(* IEC 61131-3 sources: CodesysTest/export (part 2) *)

(* ---- FB_CollectionHandlerAll.st ---- *)
FUNCTION_BLOCK FINAL FB_CollectionHandlerAll
VAR_INPUT
END_VAR
VAR
	Collection: ARRAY[0..GlobalObjects.MAX_OBJECTS] OF IAllObjects; // object array
	ObjNames   : ARRAY[0..GlobalObjects.MAX_OBJECTS] OF STRING;
	_ArrayOver   : BOOL;
	_BadObj      : INT;
	_DupeObj   : INT;
	_OverObj   : INT;
	_TotalObj   : UINT;
END_VAR

METHOD FINAL AddObject
VAR_INPUT
	Obj   : IAllObjects;
END_VAR
VAR
	AnyObject : IAllObjects;
	Fault : IFault;
	Cylinder : ICylinder;
	PositionableMotor : IPositionableMotor;
	Logger : IMachineLogger;
	Loggable : ILoggable;
	Executable : IExecuteAutomatically;
	Initializable : IInitializable;
	J   : UINT;
END_VAR
IF (__QUERYINTERFACE(Obj, AnyObject)) THEN
   // make sure haven't already added this object
   FOR J:= 1 TO _TotalObj DO
      IF Collection[J] = AnyObject THEN
         // object pointer matches - dupe!
         _DupeObj:= _DupeObj + 1;
         RETURN;
      END_IF
   END_FOR

   IF _TotalObj < GlobalObjects.MAX_OBJECTS THEN
      Collection[_TotalObj]:= AnyObject;
      ObjNames[_TotalObj]:= Obj.InstanceName;
	   _TotalObj:= _TotalObj + 1;
   ELSE
      _ArrayOver:= TRUE;
      _OverObj:= _OverObj + 1;
   END_IF
ELSE
   _BadObj:= _BadObj + 1;
END_IF

// Add object to proper collection based on its interfaces
IF (__QUERYINTERFACE(Obj, Fault)) THEN
	GlobalObjects.CollectionOfFaults.AddObject(Fault);
END_IF

IF (__QUERYINTERFACE(Obj, Cylinder)) THEN
	GlobalObjects.CollectionOfCylinders.AddObject(Cylinder);
END_IF

IF (__QUERYINTERFACE(Obj, PositionableMotor)) THEN
	GlobalObjects.CollectionOfPositionableMotors.AddObject(PositionableMotor);
END_IF

IF (__QUERYINTERFACE(Obj, Logger)) THEN
	GlobalObjects.CollectionOfLogs.AddObject(Logger);
END_IF

IF (__QUERYINTERFACE(Obj, Loggable)) THEN
	GlobalObjects.CollectionOfLoggable.AddObject(Loggable);
END_IF

IF (__QUERYINTERFACE(Obj, Executable)) THEN
	GlobalObjects.CollectionOfExecutable.AddObject(Executable);
END_IF

IF (__QUERYINTERFACE(Obj, Initializable)) THEN
	GlobalObjects.CollectionOfInitialzable.AddObject(Initializable);
END_IF

FUNCTION_BLOCK FINAL FB_CollectionHandlerAll
VAR_INPUT
END_VAR
VAR
	Collection: ARRAY[0..GlobalObjects.MAX_OBJECTS] OF IAllObjects; // object array
	ObjNames   : ARRAY[0..GlobalObjects.MAX_OBJECTS] OF STRING;
	_ArrayOver   : BOOL;
	_BadObj      : INT;
	_DupeObj   : INT;
	_OverObj   : INT;
	_TotalObj   : UINT;
END_VAR

METHOD FINAL AddObject
VAR_INPUT
	Obj   : IAllObjects;
END_VAR
VAR
	AnyObject : IAllObjects;
	Fault : IFault;
	Cylinder : ICylinder;
	PositionableMotor : IPositionableMotor;
	Logger : IMachineLogger;
	Loggable : ILoggable;
	Executable : IExecuteAutomatically;
	Initializable : IInitializable;
	J   : UINT;
END_VAR
IF (__QUERYINTERFACE(Obj, AnyObject)) THEN
   // make sure haven't already added this object
   FOR J:= 1 TO _TotalObj DO
      IF Collection[J] = AnyObject THEN
         // object pointer matches - dupe!
         _DupeObj:= _DupeObj + 1;
         RETURN;
      END_IF
   END_FOR

   IF _TotalObj < GlobalObjects.MAX_OBJECTS THEN
      Collection[_TotalObj]:= AnyObject;
      ObjNames[_TotalObj]:= Obj.InstanceName;
	   _TotalObj:= _TotalObj + 1;
   ELSE
      _ArrayOver:= TRUE;
      _OverObj:= _OverObj + 1;
   END_IF
ELSE
   _BadObj:= _BadObj + 1;
END_IF

// Add object to proper collection based on its interfaces
IF (__QUERYINTERFACE(Obj, Fault)) THEN
	GlobalObjects.CollectionOfFaults.AddObject(Fault);
END_IF

IF (__QUERYINTERFACE(Obj, Cylinder)) THEN
	GlobalObjects.CollectionOfCylinders.AddObject(Cylinder);
END_IF

IF (__QUERYINTERFACE(Obj, PositionableMotor)) THEN
	GlobalObjects.CollectionOfPositionableMotors.AddObject(PositionableMotor);
END_IF

IF (__QUERYINTERFACE(Obj, Logger)) THEN
	GlobalObjects.CollectionOfLogs.AddObject(Logger);
END_IF

IF (__QUERYINTERFACE(Obj, Loggable)) THEN
	GlobalObjects.CollectionOfLoggable.AddObject(Loggable);
END_IF

IF (__QUERYINTERFACE(Obj, Executable)) THEN
	GlobalObjects.CollectionOfExecutable.AddObject(Executable);
END_IF

IF (__QUERYINTERFACE(Obj, Initializable)) THEN
	GlobalObjects.CollectionOfInitialzable.AddObject(Initializable);
END_IF

(* ---- FB_CollectionHandlerCylinders.st ---- *)
FUNCTION_BLOCK FB_CollectionHandlerCylinders
VAR_INPUT
END_VAR
VAR
	Collection: ARRAY[0..GlobalObjects.MAX_CYLINDERS] OF ICylinder; // object array
	ObjNames   : ARRAY[0..GlobalObjects.MAX_CYLINDERS] OF STRING;
	_ArrayOver   : BOOL;
	_BadObj      : INT;
	_DupeObj   : INT;
	_OverObj   : INT;
	_TotalObj   : UINT;
END_VAR

METHOD AddObject
VAR_INPUT
	Obj   : ICylinder;
END_VAR
VAR
	Cast: ICylinder;
	J   : UINT;
END_VAR
FOR J:= 0 TO _TotalObj DO
	IF Collection[J] = Obj THEN
		// object pointer matches - dupe!
		_DupeObj:= _DupeObj + 1;
		RETURN;
	END_IF
END_FOR

IF _TotalObj < GlobalObjects.MAX_CYLINDERS THEN
	Collection[_TotalObj]:= Obj;
	ObjNames[_TotalObj]:= Obj.InstanceName;
	_TotalObj:= _TotalObj + 1;
ELSE
	_ArrayOver:= TRUE;
	_OverObj:= _OverObj + 1;
END_IF

FUNCTION_BLOCK FB_CollectionHandlerCylinders
VAR_INPUT
END_VAR
VAR
	Collection: ARRAY[0..GlobalObjects.MAX_CYLINDERS] OF ICylinder; // object array
	ObjNames   : ARRAY[0..GlobalObjects.MAX_CYLINDERS] OF STRING;
	_ArrayOver   : BOOL;
	_BadObj      : INT;
	_DupeObj   : INT;
	_OverObj   : INT;
	_TotalObj   : UINT;
END_VAR

METHOD AddObject
VAR_INPUT
	Obj   : ICylinder;
END_VAR
VAR
	Cast: ICylinder;
	J   : UINT;
END_VAR
FOR J:= 0 TO _TotalObj DO
	IF Collection[J] = Obj THEN
		// object pointer matches - dupe!
		_DupeObj:= _DupeObj + 1;
		RETURN;
	END_IF
END_FOR

IF _TotalObj < GlobalObjects.MAX_CYLINDERS THEN
	Collection[_TotalObj]:= Obj;
	ObjNames[_TotalObj]:= Obj.InstanceName;
	_TotalObj:= _TotalObj + 1;
ELSE
	_ArrayOver:= TRUE;
	_OverObj:= _OverObj + 1;
END_IF

(* ---- FB_CollectionHandlerExecutable.st ---- *)
FUNCTION_BLOCK FB_CollectionHandlerExecutable
VAR_INPUT
END_VAR
VAR
	Collection: ARRAY[0..GlobalObjects.MAX_EXECUTEABLE] OF IExecuteAutomatically; // object array
	ObjNames   : ARRAY[0..GlobalObjects.MAX_EXECUTEABLE] OF STRING;
	_ArrayOver   : BOOL;
	_BadObj      : INT;
	_DupeObj   : INT;
	_OverObj   : INT;
	_TotalObj   : UINT;
END_VAR
//	Function Block: FB_CollectionHandlerExecutable
//	Description: This collection handler stores executable FB's to an array
//				 and has a method to execute them all on demand
//	Created by: Ben Hess
//	Created Date: Friday, September 7, 2018

METHOD AddObject
VAR_INPUT
	Obj   : IExecuteAutomatically;
END_VAR
VAR
	I   : UINT;
	J : UINT;
END_VAR
// Add the active fault to the array
FOR J:= 0 TO _TotalObj DO
	IF Collection[J] = Obj THEN
		// object pointer matches - it's already in here
		RETURN;
	END_IF
END_FOR

IF _TotalObj < GlobalObjects.MAX_EXECUTEABLE THEN
	Collection[_TotalObj]:= Obj;
	ObjNames[_TotalObj]:= Obj.InstanceName;
	_TotalObj:= _TotalObj + 1;
ELSE
	_ArrayOver:= TRUE;
	_OverObj:= _OverObj + 1;
END_IF

METHOD ExecuteAll
VAR_INPUT
END_VAR
VAR
	Cast : IExecuteAutomatically;
	J : UINT;
END_VAR
// For each executable objest in the array, run its "Execute()" method
FOR J:= 0 TO _TotalObj - 1 DO
	IF (__QUERYINTERFACE(Collection[J], Cast)) THEN
		Cast.Execute();
	ELSE
		RETURN;
	END_IF
END_FOR

FUNCTION_BLOCK FB_CollectionHandlerExecutable
VAR_INPUT
END_VAR
VAR
	Collection: ARRAY[0..GlobalObjects.MAX_EXECUTEABLE] OF IExecuteAutomatically; // object array
	ObjNames   : ARRAY[0..GlobalObjects.MAX_EXECUTEABLE] OF STRING;
	_ArrayOver   : BOOL;
	_BadObj      : INT;
	_DupeObj   : INT;
	_OverObj   : INT;
	_TotalObj   : UINT;
END_VAR
//	Function Block: FB_CollectionHandlerExecutable
//	Description: This collection handler stores executable FB's to an array
//				 and has a method to execute them all on demand
//	Created by: Ben Hess
//	Created Date: Friday, September 7, 2018

METHOD AddObject
VAR_INPUT
	Obj   : IExecuteAutomatically;
END_VAR
VAR
	I   : UINT;
	J : UINT;
END_VAR
// Add the active fault to the array
FOR J:= 0 TO _TotalObj DO
	IF Collection[J] = Obj THEN
		// object pointer matches - it's already in here
		RETURN;
	END_IF
END_FOR

IF _TotalObj < GlobalObjects.MAX_EXECUTEABLE THEN
	Collection[_TotalObj]:= Obj;
	ObjNames[_TotalObj]:= Obj.InstanceName;
	_TotalObj:= _TotalObj + 1;
ELSE
	_ArrayOver:= TRUE;
	_OverObj:= _OverObj + 1;
END_IF

METHOD ExecuteAll
VAR_INPUT
END_VAR
VAR
	Cast : IExecuteAutomatically;
	J : UINT;
END_VAR
// For each executable objest in the array, run its "Execute()" method
FOR J:= 0 TO _TotalObj - 1 DO
	IF (__QUERYINTERFACE(Collection[J], Cast)) THEN
		Cast.Execute();
	ELSE
		RETURN;
	END_IF
END_FOR

(* ---- FB_CollectionHandlerFaults.st ---- *)
FUNCTION_BLOCK FB_CollectionHandlerFaults
VAR_INPUT
END_VAR
VAR
	Collection: ARRAY[0..GlobalObjects.MAX_FAULTS] OF IFault; // object array
	ObjNames   : ARRAY[0..GlobalObjects.MAX_FAULTS] OF STRING;
	faults : ARRAY[0..GlobalObjects.MAX_FAULTS] OF HMIFaultType;
	_ArrayOver   : BOOL;
	_BadObj      : INT;
	_DupeObj   : INT;
	_OverObj   : INT;
	_TotalObj   : UINT;
	_InitFaultList : BOOL;
END_VAR

METHOD FaultUpdateForHMI
VAR_INPUT
END_VAR
VAR
	I : UINT;
END_VAR
FOR I:= 0 TO _TotalObj - 1 DO
	IF NOT _InitFaultList THEN
		faults[I].name := Collection[I].InstanceName;
	END_IF
	faults[I].active := Collection[I].FaultActive;
END_FOR
_InitFaultList := TRUE;

METHOD AddObject
VAR_INPUT
	Obj   : IFault;
END_VAR
VAR
	J   : UINT;
END_VAR
FOR J:= 0 TO _TotalObj DO
	IF Collection[J] = Obj THEN
		// object pointer matches - dupe!
		_DupeObj:= _DupeObj + 1;
		RETURN;
	END_IF
END_FOR

IF _TotalObj < GlobalObjects.MAX_FAULTS THEN
	Collection[_TotalObj]:= Obj;
	ObjNames[_TotalObj]:= Obj.InstanceName;
	_TotalObj:= _TotalObj + 1;
ELSE
	_ArrayOver:= TRUE;
	_OverObj:= _OverObj + 1;
END_IF

(* ---- FB_CollectionHandlerInitializable.st ---- *)
FUNCTION_BLOCK FB_CollectionHandlerInitializable
VAR_INPUT

END_VAR
VAR
	Collection: ARRAY[0..GlobalObjects.MAX_LOGGABLE] OF IInitializable; // object array
	ObjNames   : ARRAY[0..GlobalObjects.MAX_LOGGABLE] OF STRING;
	_ArrayOver   : BOOL;
	_BadObj      : INT;
	_DupeObj   : INT;
	_OverObj   : INT;
	_TotalObj   : UINT;
END_VAR
//	Function Block: FB_CollectionHandlerLoggable
//	Description: This collection handler takes in loggable objects and registers them with a logger.  The FirstScan function should trigger the
//				 RegisterAll() method to register all loggable objects with a logger
//	Created by: Ben Hess
//	Created Date: Tuesday, September 11, 2018

METHOD AddObject
VAR_INPUT
	Obj   : IInitializable;
END_VAR
VAR
	J   : UINT;
END_VAR
FOR J:= 0 TO _TotalObj DO
	IF Collection[J] = Obj THEN
		// object pointer matches - dupe!
		_DupeObj:= _DupeObj + 1;
		RETURN;
	END_IF
END_FOR

IF _TotalObj < GlobalObjects.MAX_LOGGABLE THEN
	Collection[_TotalObj]:= Obj;
	ObjNames[_TotalObj]:= Obj.InstanceName;
	_TotalObj:= _TotalObj + 1;
ELSE
	_ArrayOver:= TRUE;
	_OverObj:= _OverObj + 1;
END_IF

METHOD InitializeAll
VAR_INPUT

END_VAR
VAR
	J : UINT;
	Cast : IInitializable;
END_VAR

FOR J:= 0 TO _TotalObj - 1 DO
	IF (__QUERYINTERFACE(Collection[J], Cast)) THEN
		Cast.Initialize();
	ELSE
		RETURN;
	END_IF
END_FOR

FUNCTION_BLOCK FB_CollectionHandlerInitializable
VAR_INPUT

END_VAR
VAR
	Collection: ARRAY[0..GlobalObjects.MAX_LOGGABLE] OF IInitializable; // object array
	ObjNames   : ARRAY[0..GlobalObjects.MAX_LOGGABLE] OF STRING;
	_ArrayOver   : BOOL;
	_BadObj      : INT;
	_DupeObj   : INT;
	_OverObj   : INT;
	_TotalObj   : UINT;
END_VAR
//	Function Block: FB_CollectionHandlerLoggable
//	Description: This collection handler takes in loggable objects and registers them with a logger.  The FirstScan function should trigger the
//				 RegisterAll() method to register all loggable objects with a logger
//	Created by: Ben Hess
//	Created Date: Tuesday, September 11, 2018

METHOD AddObject
VAR_INPUT
	Obj   : IInitializable;
END_VAR
VAR
	J   : UINT;
END_VAR
FOR J:= 0 TO _TotalObj DO
	IF Collection[J] = Obj THEN
		// object pointer matches - dupe!
		_DupeObj:= _DupeObj + 1;
		RETURN;
	END_IF
END_FOR

IF _TotalObj < GlobalObjects.MAX_LOGGABLE THEN
	Collection[_TotalObj]:= Obj;
	ObjNames[_TotalObj]:= Obj.InstanceName;
	_TotalObj:= _TotalObj + 1;
ELSE
	_ArrayOver:= TRUE;
	_OverObj:= _OverObj + 1;
END_IF

METHOD InitializeAll
VAR_INPUT

END_VAR
VAR
	J : UINT;
	Cast : IInitializable;
END_VAR

FOR J:= 0 TO _TotalObj - 1 DO
	IF (__QUERYINTERFACE(Collection[J], Cast)) THEN
		Cast.Initialize();
	ELSE
		RETURN;
	END_IF
END_FOR

(* ---- FB_CollectionHandlerLoggable.st ---- *)
FUNCTION_BLOCK FB_CollectionHandlerLoggable
VAR_INPUT

END_VAR
VAR
	Collection: ARRAY[0..GlobalObjects.MAX_LOGGABLE] OF ILoggable; // object array
	ObjNames   : ARRAY[0..GlobalObjects.MAX_LOGGABLE] OF STRING;
	_ArrayOver   : BOOL;
	_BadObj      : INT;
	_DupeObj   : INT;
	_OverObj   : INT;
	_TotalObj   : UINT;
	_internalLogger : REFERENCE TO IMachineLogger;
END_VAR
//	Function Block: FB_CollectionHandlerLoggable
//	Description: This collection handler takes in loggable objects and registers them with a logger.  The FirstScan function should trigger the
//				 RegisterAll() method to register all loggable objects with a logger
//	Created by: Ben Hess
//	Created Date: Tuesday, September 11, 2018

METHOD AddObject
VAR_INPUT
	Obj   : ILoggable;
END_VAR
VAR
	J   : UINT;
END_VAR
FOR J:= 0 TO _TotalObj DO
	IF Collection[J] = Obj THEN
		// object pointer matches - dupe!
		_DupeObj:= _DupeObj + 1;
		RETURN;
	END_IF
END_FOR

IF _TotalObj < GlobalObjects.MAX_LOGGABLE THEN
	Collection[_TotalObj]:= Obj;
	ObjNames[_TotalObj]:= Obj.InstanceName;
	_TotalObj:= _TotalObj + 1;
ELSE
	_ArrayOver:= TRUE;
	_OverObj:= _OverObj + 1;
END_IF

METHOD RegisterAll
VAR_INPUT
	internalLogger : IMachineLogger;
END_VAR
VAR
	I   : UINT;
	J : UINT;
	cast : ILoggable;
END_VAR

FOR J:= 0 TO _TotalObj - 1 DO
	IF (__QUERYINTERFACE(Collection[J], Cast)) THEN
		cast.RegisterLogger(internalLogger := internalLogger);
	ELSE
		RETURN;
	END_IF
END_FOR

FUNCTION_BLOCK FB_CollectionHandlerLoggable
VAR_INPUT

END_VAR
VAR
	Collection: ARRAY[0..GlobalObjects.MAX_LOGGABLE] OF ILoggable; // object array
	ObjNames   : ARRAY[0..GlobalObjects.MAX_LOGGABLE] OF STRING;
	_ArrayOver   : BOOL;
	_BadObj      : INT;
	_DupeObj   : INT;
	_OverObj   : INT;
	_TotalObj   : UINT;
	_internalLogger : REFERENCE TO IMachineLogger;
END_VAR
//	Function Block: FB_CollectionHandlerLoggable
//	Description: This collection handler takes in loggable objects and registers them with a logger.  The FirstScan function should trigger the
//				 RegisterAll() method to register all loggable objects with a logger
//	Created by: Ben Hess
//	Created Date: Tuesday, September 11, 2018

METHOD AddObject
VAR_INPUT
	Obj   : ILoggable;
END_VAR
VAR
	J   : UINT;
END_VAR
FOR J:= 0 TO _TotalObj DO
	IF Collection[J] = Obj THEN
		// object pointer matches - dupe!
		_DupeObj:= _DupeObj + 1;
		RETURN;
	END_IF
END_FOR

IF _TotalObj < GlobalObjects.MAX_LOGGABLE THEN
	Collection[_TotalObj]:= Obj;
	ObjNames[_TotalObj]:= Obj.InstanceName;
	_TotalObj:= _TotalObj + 1;
ELSE
	_ArrayOver:= TRUE;
	_OverObj:= _OverObj + 1;
END_IF

METHOD RegisterAll
VAR_INPUT
	internalLogger : IMachineLogger;
END_VAR
VAR
	I   : UINT;
	J : UINT;
	cast : ILoggable;
END_VAR

FOR J:= 0 TO _TotalObj - 1 DO
	IF (__QUERYINTERFACE(Collection[J], Cast)) THEN
		cast.RegisterLogger(internalLogger := internalLogger);
	ELSE
		RETURN;
	END_IF
END_FOR

(* ---- FB_CollectionHandlerLogs.st ---- *)
FUNCTION_BLOCK FB_CollectionHandlerLogs
VAR_INPUT
END_VAR
VAR
	Collection: ARRAY[0..GlobalObjects.MAX_LOGS] OF IMachineLogger; // object array
	ObjNames   : ARRAY[0..GlobalObjects.MAX_LOGS] OF STRING;
	_ArrayOver   : BOOL;
	_BadObj      : INT;
	_DupeObj   : INT;
	_OverObj   : INT;
	_TotalObj   : UINT;
END_VAR

METHOD AddObject
VAR_INPUT
	Obj   : IMachineLogger;
END_VAR
VAR
	J   : UINT;
END_VAR
FOR J:= 0 TO _TotalObj DO
	IF Collection[J] = Obj THEN
		// object pointer matches - dupe!
		_DupeObj:= _DupeObj + 1;
		RETURN;
	END_IF
END_FOR

IF _TotalObj < GlobalObjects.MAX_LOGS THEN
	Collection[_TotalObj]:= Obj;
	ObjNames[_TotalObj]:= Obj.InstanceName;
	_TotalObj:= _TotalObj + 1;
ELSE
	_ArrayOver:= TRUE;
	_OverObj:= _OverObj + 1;
END_IF

(* ---- FB_CollectionHandlerPositionableMotors.st ---- *)
FUNCTION_BLOCK FB_CollectionHandlerPositionableMotors
VAR_INPUT
END_VAR
VAR
	Collection: ARRAY[0..GlobalObjects.MAX_MOTORS] OF IPositionableMotor; // object array
	ObjNames   : ARRAY[0..GlobalObjects.MAX_MOTORS] OF STRING;
	_ArrayOver   : BOOL;
	_BadObj      : INT;
	_DupeObj   : INT;
	_OverObj   : INT;
	_TotalObj   : UINT;
END_VAR

METHOD AddObject
VAR_INPUT
	Obj   : IPositionableMotor;
END_VAR
VAR
	J   : UINT;
END_VAR
FOR J:= 0 TO _TotalObj DO
	IF Collection[J] = Obj THEN
		// object pointer matches - dupe!
		_DupeObj:= _DupeObj + 1;
		RETURN;
	END_IF
END_FOR

IF _TotalObj < GlobalObjects.MAX_MOTORS THEN
	Collection[_TotalObj]:= Obj;
	ObjNames[_TotalObj]:= Obj.InstanceName;
	_TotalObj:= _TotalObj + 1;
ELSE
	_ArrayOver:= TRUE;
	_OverObj:= _OverObj + 1;
END_IF

FUNCTION_BLOCK FB_CollectionHandlerPositionableMotors
VAR_INPUT
END_VAR
VAR
	Collection: ARRAY[0..GlobalObjects.MAX_MOTORS] OF IPositionableMotor; // object array
	ObjNames   : ARRAY[0..GlobalObjects.MAX_MOTORS] OF STRING;
	_ArrayOver   : BOOL;
	_BadObj      : INT;
	_DupeObj   : INT;
	_OverObj   : INT;
	_TotalObj   : UINT;
END_VAR

METHOD AddObject
VAR_INPUT
	Obj   : IPositionableMotor;
END_VAR
VAR
	J   : UINT;
END_VAR
FOR J:= 0 TO _TotalObj DO
	IF Collection[J] = Obj THEN
		// object pointer matches - dupe!
		_DupeObj:= _DupeObj + 1;
		RETURN;
	END_IF
END_FOR

IF _TotalObj < GlobalObjects.MAX_MOTORS THEN
	Collection[_TotalObj]:= Obj;
	ObjNames[_TotalObj]:= Obj.InstanceName;
	_TotalObj:= _TotalObj + 1;
ELSE
	_ArrayOver:= TRUE;
	_OverObj:= _OverObj + 1;
END_IF

(* ---- FB_Delay.st ---- *)
FUNCTION_BLOCK FB_Delay IMPLEMENTS IExecuteAutomatically
VAR_INPUT
	in : BOOL;
	delay : TIME;
END_VAR
VAR_OUTPUT
	Q : BOOL;
END_VAR
VAR
	delayTimer : TON;
END_VAR

METHOD Execute

delayTimer(IN := in, PT := delay, Q => Q);

FUNCTION_BLOCK FB_Delay IMPLEMENTS IExecuteAutomatically
VAR_INPUT
	in : BOOL;
	delay : TIME;
END_VAR
VAR_OUTPUT
	Q : BOOL;
END_VAR
VAR
	delayTimer : TON;
END_VAR

METHOD Execute

delayTimer(IN := in, PT := delay, Q => Q);

(* ---- FB_DoubleSolenoidClosedCenterActuator.st ---- *)
FUNCTION_BLOCK FB_DoubleSolenoidClosedCenterActuator EXTENDS FB_PneumaticActuator IMPLEMENTS IExtendLowPressure
VAR_INPUT
END_VAR
VAR_OUTPUT
END_VAR
VAR

END_VAR

PROPERTY ExtendAsserted : BOOL

PROPERTY RetractAsserted : BOOL

METHOD Extend

THIS^.solenoid0 := TRUE;
THIS^.solenoid1 := FALSE;

METHOD Retract

THIS^.solenoid0 := FALSE;
THIS^.solenoid1 := TRUE;

METHOD ExtendLowPressure
VAR_INPUT
END_VAR

THIS^.solenoid0 := TRUE;
THIS^.solenoid1 := TRUE;

PROPERTY ExtendLPAsserted : BOOL

FUNCTION_BLOCK FB_DoubleSolenoidClosedCenterActuator EXTENDS FB_PneumaticActuator IMPLEMENTS IExtendLowPressure
VAR_INPUT
END_VAR
VAR_OUTPUT
END_VAR
VAR

END_VAR

PROPERTY ExtendAsserted : BOOL

PROPERTY RetractAsserted : BOOL

METHOD Extend

THIS^.solenoid0 := TRUE;
THIS^.solenoid1 := FALSE;

METHOD Retract

THIS^.solenoid0 := FALSE;
THIS^.solenoid1 := TRUE;

METHOD ExtendLowPressure
VAR_INPUT
END_VAR

THIS^.solenoid0 := TRUE;
THIS^.solenoid1 := TRUE;

PROPERTY ExtendLPAsserted : BOOL

(* ---- FB_DoubleSolenoidClosedCenterActuator_UnitTests.st ---- *)
(*
*)
{attribute 'test' := 'multitest'}
{attribute 'testcasename':='Double Solenoid Closed Center'}
{attribute 'testcategory':='Solenoids'}
{attribute 'testcasetimeout':='15000'}
FUNCTION_BLOCK FB_DoubleSolenoidClosedCenterActuator_UnitTests EXTENDS CBM.EtrigA
VAR_INPUT
	xGetTestInfo : BOOL;
    diTestCaseIndex : DINT;
END_VAR
VAR_OUTPUT
    sTestCaseName : STRING;
	sTestCaseCategories : STRING;
    diTestCaseCount : DINT;
    diTestCaseTimeout : DINT;
    sInfo : STRING;
	eError : UnitTestErrors;
    sError : STRING;
    eFailureMode : TM.FAILUREMODE;
END_VAR
VAR
	testee : FB_DoubleSolenoidClosedCenterActuator(name := 'Unit Test Actuator');
END_VAR
SUPER^();

{attribute 'hide'}
METHOD prvAbort : BOOL

SUPER^.prvAbort();

xAbortInProgress := FALSE;

{attribute 'hide'}
METHOD prvCyclicAction : BOOL

SUPER^.prvCyclicAction();
THIS^.diTestCaseCount := 4;

CASE diTestCaseIndex OF
    0: // Test Case #0
        IF THIS^.xGetTestInfo THEN
            THIS^.sTestCaseName := 'Step 1: Test Solonoids Off';
            THIS^.sTestCaseCategories := 'Solenoids';
            THIS^.diTestCaseTimeout := 3000;
			xDone := TRUE;
		ELSE
			IF NOT testee.Solenoid0Asserted AND NOT testee.Solenoid1Asserted THEN
				 xDone := TRUE;
			ELSE
				THIS^.sError := 'Solenoids not off';
				xError := TRUE;
				eError := UnitTestErrors.Failure;
            	eFailureMode := TM.FAILUREMODE.AbortTestCase;
                iError := 1;
			END_IF
        END_IF
    1: // Test Case #1
        IF THIS^.xGetTestInfo THEN
            THIS^.sTestCaseName := 'Step 2: Extend Cylinder';
            THIS^.sTestCaseCategories := 'Solenoids';
            THIS^.diTestCaseTimeout := 3000;
            xDone := TRUE;
		ELSE
			testee.Extend();
			IF testee.Solenoid0Asserted AND testee.ExtendAsserted
				AND NOT testee.Solenoid1Asserted AND NOT testee.RetractAsserted THEN
				 xDone := TRUE;
			ELSE
				THIS^.sError := 'Failed to extend';
				xError := TRUE;
				eError := UnitTestErrors.Failure;
            	eFailureMode := TM.FAILUREMODE.AbortTestCase;
                iError := 2;
			END_IF
       END_IF

	2:	//
		IF THIS^.xGetTestInfo THEN
            THIS^.sTestCaseName := 'Step 3: Retract Cylinder';
            THIS^.sTestCaseCategories := 'Solenoids';
            THIS^.diTestCaseTimeout := 3000;
            xDone := TRUE;
		ELSE
			testee.Retract();
			IF testee.Solenoid1Asserted AND testee.RetractAsserted
				AND NOT testee.Solenoid0Asserted AND NOT testee.ExtendAsserted THEN
				 xDone := TRUE;
			ELSE
				THIS^.sError := 'Failed to retract';
				xError := TRUE;
				eError := UnitTestErrors.Failure;
            	eFailureMode := TM.FAILUREMODE.AbortTestCase;
                iError := 3;
			END_IF
       END_IF

   	3:	IF THIS^.xGetTestInfo THEN
            THIS^.sTestCaseName := 'Step 4: Extend Low Pressure';
            THIS^.sTestCaseCategories := 'Solenoids';
            THIS^.diTestCaseTimeout := 3000;
            xDone := TRUE;
		ELSE
			testee.ExtendLowPressure();
			IF testee.Solenoid1Asserted AND testee.ExtendLPAsserted
				AND testee.Solenoid0Asserted
				AND NOT testee.RetractAsserted THEN
				 xDone := TRUE;
			ELSE
				THIS^.sError := 'Failed to extend low pressure';
				xError := TRUE;
				eError := UnitTestErrors.Failure;
            	eFailureMode := TM.FAILUREMODE.AbortTestCase;
                iError := 3;
			END_IF
       END_IF
    ELSE
        IF THIS^.diTestCaseIndex < 0 THEN
            THIS^.diTestCaseCount := 4;
            xDone := TRUE;
        ELSE
            THIS^.sInfo := 'Invalid test case index';
            eError := UnitTestErrors.Failure;
			xError := TRUE;
        END_IF
END_CASE

{attribute 'hide'}
METHOD prvResetOutputs : BOOL

SUPER^.prvResetOutputs();

sTestCaseName := '';
sTestCaseCategories := '';
diTestCaseCount := 0;
diTestCaseTimeout := 0;
sInfo := '';
sError := '';
eFailureMode := TM.FAILUREMODE.AbortTestCase;

{attribute 'hide'}
METHOD prvStart : BOOL

SUPER^.prvStart();

(*
*)
{attribute 'test' := 'multitest'}
{attribute 'testcasename':='Double Solenoid Closed Center'}
{attribute 'testcategory':='Solenoids'}
{attribute 'testcasetimeout':='15000'}
FUNCTION_BLOCK FB_DoubleSolenoidClosedCenterActuator_UnitTests EXTENDS CBM.EtrigA
VAR_INPUT
	xGetTestInfo : BOOL;
    diTestCaseIndex : DINT;
END_VAR
VAR_OUTPUT
    sTestCaseName : STRING;
	sTestCaseCategories : STRING;
    diTestCaseCount : DINT;
    diTestCaseTimeout : DINT;
    sInfo : STRING;
	eError : UnitTestErrors;
    sError : STRING;
    eFailureMode : TM.FAILUREMODE;
END_VAR
VAR
	testee : FB_DoubleSolenoidClosedCenterActuator(name := 'Unit Test Actuator');
END_VAR
SUPER^();

{attribute 'hide'}
METHOD prvAbort : BOOL

SUPER^.prvAbort();

xAbortInProgress := FALSE;

{attribute 'hide'}
METHOD prvCyclicAction : BOOL

SUPER^.prvCyclicAction();
THIS^.diTestCaseCount := 4;

CASE diTestCaseIndex OF
    0: // Test Case #0
        IF THIS^.xGetTestInfo THEN
            THIS^.sTestCaseName := 'Step 1: Test Solonoids Off';
            THIS^.sTestCaseCategories := 'Solenoids';
            THIS^.diTestCaseTimeout := 3000;
			xDone := TRUE;
		ELSE
			IF NOT testee.Solenoid0Asserted AND NOT testee.Solenoid1Asserted THEN
				 xDone := TRUE;
			ELSE
				THIS^.sError := 'Solenoids not off';
				xError := TRUE;
				eError := UnitTestErrors.Failure;
            	eFailureMode := TM.FAILUREMODE.AbortTestCase;
                iError := 1;
			END_IF
        END_IF
    1: // Test Case #1
        IF THIS^.xGetTestInfo THEN
            THIS^.sTestCaseName := 'Step 2: Extend Cylinder';
            THIS^.sTestCaseCategories := 'Solenoids';
            THIS^.diTestCaseTimeout := 3000;
            xDone := TRUE;
		ELSE
			testee.Extend();
			IF testee.Solenoid0Asserted AND testee.ExtendAsserted
				AND NOT testee.Solenoid1Asserted AND NOT testee.RetractAsserted THEN
				 xDone := TRUE;
			ELSE
				THIS^.sError := 'Failed to extend';
				xError := TRUE;
				eError := UnitTestErrors.Failure;
            	eFailureMode := TM.FAILUREMODE.AbortTestCase;
                iError := 2;
			END_IF
       END_IF

	2:	//
		IF THIS^.xGetTestInfo THEN
            THIS^.sTestCaseName := 'Step 3: Retract Cylinder';
            THIS^.sTestCaseCategories := 'Solenoids';
            THIS^.diTestCaseTimeout := 3000;
            xDone := TRUE;
		ELSE
			testee.Retract();
			IF testee.Solenoid1Asserted AND testee.RetractAsserted
				AND NOT testee.Solenoid0Asserted AND NOT testee.ExtendAsserted THEN
				 xDone := TRUE;
			ELSE
				THIS^.sError := 'Failed to retract';
				xError := TRUE;
				eError := UnitTestErrors.Failure;
            	eFailureMode := TM.FAILUREMODE.AbortTestCase;
                iError := 3;
			END_IF
       END_IF

   	3:	IF THIS^.xGetTestInfo THEN
            THIS^.sTestCaseName := 'Step 4: Extend Low Pressure';
            THIS^.sTestCaseCategories := 'Solenoids';
            THIS^.diTestCaseTimeout := 3000;
            xDone := TRUE;
		ELSE
			testee.ExtendLowPressure();
			IF testee.Solenoid1Asserted AND testee.ExtendLPAsserted
				AND testee.Solenoid0Asserted
				AND NOT testee.RetractAsserted THEN
				 xDone := TRUE;
			ELSE
				THIS^.sError := 'Failed to extend low pressure';
				xError := TRUE;
				eError := UnitTestErrors.Failure;
            	eFailureMode := TM.FAILUREMODE.AbortTestCase;
                iError := 3;
			END_IF
       END_IF
    ELSE
        IF THIS^.diTestCaseIndex < 0 THEN
            THIS^.diTestCaseCount := 4;
            xDone := TRUE;
        ELSE
            THIS^.sInfo := 'Invalid test case index';
            eError := UnitTestErrors.Failure;
			xError := TRUE;
        END_IF
END_CASE

{attribute 'hide'}
METHOD prvResetOutputs : BOOL

SUPER^.prvResetOutputs();

sTestCaseName := '';
sTestCaseCategories := '';
diTestCaseCount := 0;
diTestCaseTimeout := 0;
sInfo := '';
sError := '';
eFailureMode := TM.FAILUREMODE.AbortTestCase;

{attribute 'hide'}
METHOD prvStart : BOOL

SUPER^.prvStart();

(* ---- FB_DoubleSolenoidOpenCenterActuator.st ---- *)
FUNCTION_BLOCK FINAL FB_DoubleSolenoidOpenCenterActuator EXTENDS FB_DoubleSolenoidClosedCenterActuator IMPLEMENTS IExhaustable
VAR_INPUT
END_VAR
VAR_OUTPUT
END_VAR
VAR
END_VAR

METHOD Exhaust : BOOL

THIS^.solenoid0 := FALSE;
THIS^.solenoid1 := FALSE;

FUNCTION_BLOCK FINAL FB_DoubleSolenoidOpenCenterActuator EXTENDS FB_DoubleSolenoidClosedCenterActuator IMPLEMENTS IExhaustable
VAR_INPUT
END_VAR
VAR_OUTPUT
END_VAR
VAR
END_VAR

METHOD Exhaust : BOOL

THIS^.solenoid0 := FALSE;
THIS^.solenoid1 := FALSE;

(* ---- FB_DoubleSolenoidOpenCenterActuator_UnitTests.st ---- *)
(*
*)
{attribute 'test' := 'multitest'}
{attribute 'testcasename':='Double Solenoid Open Center'}
{attribute 'testcategory':='Solenoids'}
{attribute 'testcasetimeout':='15000'}
FUNCTION_BLOCK FB_DoubleSolenoidOpenCenterActuator_UnitTests EXTENDS CBM.EtrigA
VAR_INPUT
	xGetTestInfo : BOOL;
    diTestCaseIndex : DINT;
END_VAR
VAR_OUTPUT
    sTestCaseName : STRING;
	sTestCaseCategories : STRING;
    diTestCaseCount : DINT;
    diTestCaseTimeout : DINT;
    sInfo : STRING;
	eError : UnitTestErrors;
    sError : STRING;
    eFailureMode : TM.FAILUREMODE;
END_VAR
VAR
	testee : FB_DoubleSolenoidOpenCenterActuator(name := 'Unit Test Actuator');
END_VAR
SUPER^();

{attribute 'hide'}
METHOD prvAbort : BOOL

SUPER^.prvAbort();

xAbortInProgress := FALSE;

{attribute 'hide'}
METHOD prvCyclicAction : BOOL

SUPER^.prvCyclicAction();
THIS^.diTestCaseCount := 5;

CASE diTestCaseIndex OF
    0: // Test Case #0
        IF THIS^.xGetTestInfo THEN
            THIS^.sTestCaseName := 'Step 1: Test Solonoids Off';
            THIS^.sTestCaseCategories := 'Solenoids';
            THIS^.diTestCaseTimeout := 3000;
			xDone := TRUE;
		ELSE
			IF NOT testee.Solenoid0Asserted AND NOT testee.Solenoid1Asserted THEN
				 xDone := TRUE;
			ELSE
				THIS^.sError := 'Solenoids not off';
				xError := TRUE;
				eError := UnitTestErrors.Failure;
            	eFailureMode := TM.FAILUREMODE.AbortTestCase;
                iError := 1;
			END_IF
        END_IF
    1: // Test Case #1
        IF THIS^.xGetTestInfo THEN
            THIS^.sTestCaseName := 'Step 2: Extend Cylinder';
            THIS^.sTestCaseCategories := 'Solenoids';
            THIS^.diTestCaseTimeout := 3000;
            xDone := TRUE;
		ELSE
			testee.Extend();
			IF testee.Solenoid0Asserted AND testee.ExtendAsserted
				AND NOT testee.Solenoid1Asserted AND NOT testee.RetractAsserted THEN
				 xDone := TRUE;
			ELSE
				THIS^.sError := 'Failed to extend';
				xError := TRUE;
				eError := UnitTestErrors.Failure;
            	eFailureMode := TM.FAILUREMODE.AbortTestCase;
                iError := 2;
			END_IF
       END_IF

	2:	//
		IF THIS^.xGetTestInfo THEN
            THIS^.sTestCaseName := 'Step 3: Retract Cylinder';
            THIS^.sTestCaseCategories := 'Solenoids';
            THIS^.diTestCaseTimeout := 3000;
            xDone := TRUE;
		ELSE
			testee.Retract();
			IF testee.Solenoid1Asserted AND testee.RetractAsserted
				AND NOT testee.Solenoid0Asserted AND NOT testee.ExtendAsserted THEN
				 xDone := TRUE;
			ELSE
				THIS^.sError := 'Failed to retract';
				xError := TRUE;
				eError := UnitTestErrors.Failure;
            	eFailureMode := TM.FAILUREMODE.AbortTestCase;
                iError := 3;
			END_IF
       END_IF

   	3:	IF THIS^.xGetTestInfo THEN
            THIS^.sTestCaseName := 'Step 4: Extend Low Pressure';
            THIS^.sTestCaseCategories := 'Solenoids';
            THIS^.diTestCaseTimeout := 3000;
            xDone := TRUE;
		ELSE
			testee.ExtendLowPressure();
			IF testee.Solenoid1Asserted AND testee.ExtendLPAsserted
				AND testee.Solenoid0Asserted
				AND NOT testee.RetractAsserted THEN
				 xDone := TRUE;
			ELSE
				THIS^.sError := 'Failed to extend low pressure';
				xError := TRUE;
				eError := UnitTestErrors.Failure;
            	eFailureMode := TM.FAILUREMODE.AbortTestCase;
                iError := 3;
			END_IF
       END_IF

	4: // Test Case #4
        IF THIS^.xGetTestInfo THEN
            THIS^.sTestCaseName := 'Step 5: Test Exhaust';
            THIS^.sTestCaseCategories := 'Solenoids';
            THIS^.diTestCaseTimeout := 3000;
			xDone := TRUE;
		ELSE
			testee.Exhaust();
			IF NOT testee.Solenoid0Asserted AND NOT testee.Solenoid1Asserted
				AND NOT testee.ExtendAsserted AND NOT testee.RetractAsserted THEN
				 xDone := TRUE;
			ELSE
				THIS^.sError := 'Solenoids not off';
				xError := TRUE;
				eError := UnitTestErrors.Failure;
            	eFailureMode := TM.FAILUREMODE.AbortTestCase;
                iError := 1;
			END_IF
        END_IF
    ELSE
        IF THIS^.diTestCaseIndex < 0 THEN
            THIS^.diTestCaseCount := 5;
            xDone := TRUE;
        ELSE
            THIS^.sInfo := 'Invalid test case index';
            eError := UnitTestErrors.Failure;
			xError := TRUE;
        END_IF
END_CASE

{attribute 'hide'}
METHOD prvResetOutputs : BOOL

SUPER^.prvResetOutputs();

sTestCaseName := '';
sTestCaseCategories := '';
diTestCaseCount := 0;
diTestCaseTimeout := 0;
sInfo := '';
sError := '';
eFailureMode := TM.FAILUREMODE.AbortTestCase;

{attribute 'hide'}
METHOD prvStart : BOOL

SUPER^.prvStart();

(*
*)
{attribute 'test' := 'multitest'}
{attribute 'testcasename':='Double Solenoid Open Center'}
{attribute 'testcategory':='Solenoids'}
{attribute 'testcasetimeout':='15000'}
FUNCTION_BLOCK FB_DoubleSolenoidOpenCenterActuator_UnitTests EXTENDS CBM.EtrigA
VAR_INPUT
	xGetTestInfo : BOOL;
    diTestCaseIndex : DINT;
END_VAR
VAR_OUTPUT
    sTestCaseName : STRING;
	sTestCaseCategories : STRING;
    diTestCaseCount : DINT;
    diTestCaseTimeout : DINT;
    sInfo : STRING;
	eError : UnitTestErrors;
    sError : STRING;
    eFailureMode : TM.FAILUREMODE;
END_VAR
VAR
	testee : FB_DoubleSolenoidOpenCenterActuator(name := 'Unit Test Actuator');
END_VAR
SUPER^();

{attribute 'hide'}
METHOD prvAbort : BOOL

SUPER^.prvAbort();

xAbortInProgress := FALSE;

{attribute 'hide'}
METHOD prvCyclicAction : BOOL

SUPER^.prvCyclicAction();
THIS^.diTestCaseCount := 5;

CASE diTestCaseIndex OF
    0: // Test Case #0
        IF THIS^.xGetTestInfo THEN
            THIS^.sTestCaseName := 'Step 1: Test Solonoids Off';
            THIS^.sTestCaseCategories := 'Solenoids';
            THIS^.diTestCaseTimeout := 3000;
			xDone := TRUE;
		ELSE
			IF NOT testee.Solenoid0Asserted AND NOT testee.Solenoid1Asserted THEN
				 xDone := TRUE;
			ELSE
				THIS^.sError := 'Solenoids not off';
				xError := TRUE;
				eError := UnitTestErrors.Failure;
            	eFailureMode := TM.FAILUREMODE.AbortTestCase;
                iError := 1;
			END_IF
        END_IF
    1: // Test Case #1
        IF THIS^.xGetTestInfo THEN
            THIS^.sTestCaseName := 'Step 2: Extend Cylinder';
            THIS^.sTestCaseCategories := 'Solenoids';
            THIS^.diTestCaseTimeout := 3000;
            xDone := TRUE;
		ELSE
			testee.Extend();
			IF testee.Solenoid0Asserted AND testee.ExtendAsserted
				AND NOT testee.Solenoid1Asserted AND NOT testee.RetractAsserted THEN
				 xDone := TRUE;
			ELSE
				THIS^.sError := 'Failed to extend';
				xError := TRUE;
				eError := UnitTestErrors.Failure;
            	eFailureMode := TM.FAILUREMODE.AbortTestCase;
                iError := 2;
			END_IF
       END_IF

	2:	//
		IF THIS^.xGetTestInfo THEN
            THIS^.sTestCaseName := 'Step 3: Retract Cylinder';
            THIS^.sTestCaseCategories := 'Solenoids';
            THIS^.diTestCaseTimeout := 3000;
            xDone := TRUE;
		ELSE
			testee.Retract();
			IF testee.Solenoid1Asserted AND testee.RetractAsserted
				AND NOT testee.Solenoid0Asserted AND NOT testee.ExtendAsserted THEN
				 xDone := TRUE;
			ELSE
				THIS^.sError := 'Failed to retract';
				xError := TRUE;
				eError := UnitTestErrors.Failure;
            	eFailureMode := TM.FAILUREMODE.AbortTestCase;
                iError := 3;
			END_IF
       END_IF

   	3:	IF THIS^.xGetTestInfo THEN
            THIS^.sTestCaseName := 'Step 4: Extend Low Pressure';
            THIS^.sTestCaseCategories := 'Solenoids';
            THIS^.diTestCaseTimeout := 3000;
            xDone := TRUE;
		ELSE
			testee.ExtendLowPressure();
			IF testee.Solenoid1Asserted AND testee.ExtendLPAsserted
				AND testee.Solenoid0Asserted
				AND NOT testee.RetractAsserted THEN
				 xDone := TRUE;
			ELSE
				THIS^.sError := 'Failed to extend low pressure';
				xError := TRUE;
				eError := UnitTestErrors.Failure;
            	eFailureMode := TM.FAILUREMODE.AbortTestCase;
                iError := 3;
			END_IF
       END_IF

	4: // Test Case #4
        IF THIS^.xGetTestInfo THEN
            THIS^.sTestCaseName := 'Step 5: Test Exhaust';
            THIS^.sTestCaseCategories := 'Solenoids';
            THIS^.diTestCaseTimeout := 3000;
			xDone := TRUE;
		ELSE
			testee.Exhaust();
			IF NOT testee.Solenoid0Asserted AND NOT testee.Solenoid1Asserted
				AND NOT testee.ExtendAsserted AND NOT testee.RetractAsserted THEN
				 xDone := TRUE;
			ELSE
				THIS^.sError := 'Solenoids not off';
				xError := TRUE;
				eError := UnitTestErrors.Failure;
            	eFailureMode := TM.FAILUREMODE.AbortTestCase;
                iError := 1;
			END_IF
        END_IF
    ELSE
        IF THIS^.diTestCaseIndex < 0 THEN
            THIS^.diTestCaseCount := 5;
            xDone := TRUE;
        ELSE
            THIS^.sInfo := 'Invalid test case index';
            eError := UnitTestErrors.Failure;
			xError := TRUE;
        END_IF
END_CASE

{attribute 'hide'}
METHOD prvResetOutputs : BOOL

SUPER^.prvResetOutputs();

sTestCaseName := '';
sTestCaseCategories := '';
diTestCaseCount := 0;
diTestCaseTimeout := 0;
sInfo := '';
sError := '';
eFailureMode := TM.FAILUREMODE.AbortTestCase;

{attribute 'hide'}
METHOD prvStart : BOOL

SUPER^.prvStart();

(* ---- FB_Fault.st ---- *)
FUNCTION_BLOCK FINAL FB_Fault EXTENDS FB_BaseObject IMPLEMENTS IFault, ILoggable, IExecuteAutomatically
VAR_INPUT
	ackCommand : BOOL;
	faultTrigger : BOOL;
END_VAR
VAR_OUTPUT
	acknowledged : BOOL;
	Active : BOOL;
END_VAR
VAR
	_active : BOOL;
	_acked : BOOL;
	_ackCommand : BOOL;
	ackCommandOSR : R_TRIG;
	faultTriggerONS : FB_ONS;
	activeONS : FB_ONS;
END_VAR
VAR_IN_OUT

END_VAR

METHOD Ack
IF _ackCommand OR _acked THEN
	RETURN;
END_IF
_acked := TRUE;
// Log the ACK.
_logger.AddLogItem(CONCAT(InstanceName,  ' Acked'));

METHOD Execute

//	Function Block: FB_Fault
//	Description: Faults should be of this FB type.
//  An associated FaultType variable needs to be declared in the HMIData global variable list in order to be exposed via OPCUA
//	Implementation should look as follows:
//
//  *** Instantiate the fault with constructor that contains the fault name: ***
//  VAR (*Faults*)
//		exampleFault1 : FB_Fault(name := CONCAT(_prefix,  'Example Fault 1'));
//		exampleFault2 : FB_Fault(name := CONCAT(_prefix,  'Example Fault 2'));
//  END_VAR
//
//  *** In alarm area of FB call the fault(s). refHMIFaults is passed in from above***
//  IF __ISVALIDREF(refHMIFaults) THEN
//		exampleFault1(HMIFault := refHMIFaults.exampleFault1);
//		exampleFault2(HMIFault := refHMIFaults.exampleFault2, faultTrigger := someFaultCondition);
//  END_IF
//
//	*** Either assign faultTrigger in call (as in exampleFault2 above) or set it later in logic
//	exampleFault1.faultTrigger := someFaultCondition;
//
//	Created by: Ben Hess
//	Created Date: Tuesday, May 22, 2018

ackCommandOSR(CLK := _ackCommand);
faultTriggerONS(CLK := faultTrigger);
activeONS(CLK := _active);

IF faultTriggerONS.OSR THEN
	Trigger();
END_IF

IF ackCommandOSR.Q THEN
	_acked := TRUE;
	_ackCommand := FALSE;
END_IF

IF _acked AND NOT faultTrigger THEN
	_active := FALSE;
	_acked := FALSE;
END_IF

IF activeONS.OSF THEN
	GlobalObjects.CollectionOfActiveFaults.RemoveObject(THIS^);
	_logger.AddLogItem(CONCAT(InstanceName, ' Cleared'));
END_IF

// The following is for external communication to HMI etc.
IF ackCommand THEN
	Ack();
	ackCommand := FALSE;
END_IF
Active := _active;
acknowledged := _acked;

PROPERTY InstanceName : STRING

METHOD RegisterLogger
VAR_INPUT
	internalLogger : IMachineLogger;
END_VAR

_logger := internalLogger;

METHOD Trigger

IF _active = TRUE THEN
	RETURN;
END_IF
_active := TRUE;
GlobalObjects.CollectionOfActiveFaults.AddObject(THIS^);
_logger.AddLogItem(CONCAT(InstanceName,  ' Active'));

{attribute 'monitoring' := 'variable'}
PROPERTY FaultActive : BOOL

FUNCTION_BLOCK FINAL FB_Fault EXTENDS FB_BaseObject IMPLEMENTS IFault, ILoggable, IExecuteAutomatically
VAR_INPUT
	ackCommand : BOOL;
	faultTrigger : BOOL;
END_VAR
VAR_OUTPUT
	acknowledged : BOOL;
	Active : BOOL;
END_VAR
VAR
	_active : BOOL;
	_acked : BOOL;
	_ackCommand : BOOL;
	ackCommandOSR : R_TRIG;
	faultTriggerONS : FB_ONS;
	activeONS : FB_ONS;
END_VAR
VAR_IN_OUT

END_VAR

METHOD Ack
IF _ackCommand OR _acked THEN
	RETURN;
END_IF
_acked := TRUE;
// Log the ACK.
_logger.AddLogItem(CONCAT(InstanceName,  ' Acked'));

METHOD Execute

//	Function Block: FB_Fault
//	Description: Faults should be of this FB type.
//  An associated FaultType variable needs to be declared in the HMIData global variable list in order to be exposed via OPCUA
//	Implementation should look as follows:
//
//  *** Instantiate the fault with constructor that contains the fault name: ***
//  VAR (*Faults*)
//		exampleFault1 : FB_Fault(name := CONCAT(_prefix,  'Example Fault 1'));
//		exampleFault2 : FB_Fault(name := CONCAT(_prefix,  'Example Fault 2'));
//  END_VAR
//
//  *** In alarm area of FB call the fault(s). refHMIFaults is passed in from above***
//  IF __ISVALIDREF(refHMIFaults) THEN
//		exampleFault1(HMIFault := refHMIFaults.exampleFault1);
//		exampleFault2(HMIFault := refHMIFaults.exampleFault2, faultTrigger := someFaultCondition);
//  END_IF
//
//	*** Either assign faultTrigger in call (as in exampleFault2 above) or set it later in logic
//	exampleFault1.faultTrigger := someFaultCondition;
//
//	Created by: Ben Hess
//	Created Date: Tuesday, May 22, 2018

ackCommandOSR(CLK := _ackCommand);
faultTriggerONS(CLK := faultTrigger);
activeONS(CLK := _active);

IF faultTriggerONS.OSR THEN
	Trigger();
END_IF

IF ackCommandOSR.Q THEN
	_acked := TRUE;
	_ackCommand := FALSE;
END_IF

IF _acked AND NOT faultTrigger THEN
	_active := FALSE;
	_acked := FALSE;
END_IF

IF activeONS.OSF THEN
	GlobalObjects.CollectionOfActiveFaults.RemoveObject(THIS^);
	_logger.AddLogItem(CONCAT(InstanceName, ' Cleared'));
END_IF

// The following is for external communication to HMI etc.
IF ackCommand THEN
	Ack();
	ackCommand := FALSE;
END_IF
Active := _active;
acknowledged := _acked;

PROPERTY InstanceName : STRING

METHOD RegisterLogger
VAR_INPUT
	internalLogger : IMachineLogger;
END_VAR

_logger := internalLogger;

METHOD Trigger

IF _active = TRUE THEN
	RETURN;
END_IF
_active := TRUE;
GlobalObjects.CollectionOfActiveFaults.AddObject(THIS^);
_logger.AddLogItem(CONCAT(InstanceName,  ' Active'));

{attribute 'monitoring' := 'variable'}
PROPERTY FaultActive : BOOL

(* ---- FB_Fault_Test.st ---- *)
{attribute 'test' := 'multitest'}
{attribute 'testcasename':='Fault FB'}
{attribute 'testcategory':='Basics'}
{attribute 'testcasetimeout':='5000'}
FUNCTION_BLOCK FB_Fault_Test EXTENDS TM.Testcase_Base
VAR_INPUT
     xGetTestInfo : BOOL;
    diTestCaseIndex : DINT;
END_VAR
VAR_OUTPUT
   sTestCaseName : STRING;
    sTestCaseCategories : STRING;
    diTestCaseCount : DINT;
    diTestCaseTimeout : DINT;
    sInfo : STRING;
    eError : FB_Fault_Test_Errors;
    sError : STRING;
    eFailureMode : TM.FAILUREMODE;
END_VAR
VAR
	faultToTest : FB_Fault(name := 'Test Fault');
END_VAR

SUPER^();

{attribute 'hide'}
METHOD prvAbort : BOOL

SUPER^.prvAbort();

xAbortInProgress := FALSE;

{attribute 'hide'}
METHOD prvCyclicAction : BOOL

SUPER^.prvCyclicAction();
faultToTest.Execute();
THIS^.diTestCaseCount := 3;
CASE diTestCaseIndex OF
    0: // Test Case #0
        IF THIS^.xGetTestInfo THEN
            THIS^.sTestCaseName := 'Step 1: Check Fault is not active';
            THIS^.sTestCaseCategories := 'General';
            THIS^.diTestCaseTimeout := 3000;
			xDone := TRUE;
		ELSE
			IF NOT faultToTest.FaultActive THEN
				 xDone := TRUE;
			ELSE
				THIS^.sError := 'Fault Active before Trigger';
				xError := TRUE;
				eError := FB_Fault_Test_Errors.Fault_Active;
            	eFailureMode := TM.FAILUREMODE.AbortTestCase;
                iError := 1;
			END_IF
        END_IF
    1: // Test Case #1
        IF THIS^.xGetTestInfo THEN
            THIS^.sTestCaseName := 'Step 2: Trigger Fault';
            THIS^.sTestCaseCategories := 'General';
            THIS^.diTestCaseTimeout := 3000;
            xDone := TRUE;
		ELSE
			faultToTest.Trigger();
			IF faultToTest.FaultActive THEN
				 xDone := TRUE;
			ELSE
				THIS^.sError := 'Fault Failed to Trigger';
				xError := TRUE;
				eError := FB_Fault_Test_Errors.Fault_Not_Triggered;
				eFailureMode := TM.FAILUREMODE.AbortTestCase;
                iError := 2;
			END_IF
       END_IF

	2:	//
		IF THIS^.xGetTestInfo THEN
            THIS^.sTestCaseName := 'Step 3: Reset Fault';
            THIS^.sTestCaseCategories := 'General';
            THIS^.diTestCaseTimeout := 3000;
            xDone := TRUE;
		ELSE
			faultToTest.Ack();
			faultToTest.Execute();
			IF NOT faultToTest.FaultActive THEN
				 xDone := TRUE;
			ELSE
				THIS^.sError := 'Fault did not reset';
				xError := TRUE;
				eError := FB_Fault_Test_Errors.Fault_Not_Reset;
				eFailureMode := TM.FAILUREMODE.AbortTestCase;
                iError := 3;
			END_IF
       END_IF

    ELSE
        IF THIS^.diTestCaseIndex < 0 THEN
            THIS^.diTestCaseCount := 3;
            xDone := TRUE;
        ELSE
            THIS^.sInfo := 'Invalid test case index';
            eError := FB_Fault_Test_Errors.Fault_Not_Reset;
			xError := TRUE;
        END_IF
END_CASE

{attribute 'hide'}
METHOD prvResetOutputs : BOOL

SUPER^.prvResetOutputs();

sTestCaseName := '';
sTestCaseCategories := '';
diTestCaseCount := 0;
diTestCaseTimeout := 0;
sInfo := '';
sError := '';
eFailureMode := TM.FAILUREMODE.AbortTestCase;
eError := FB_Fault_Test_Errors.No_Error;

{attribute 'hide'}
{warning 'Add method implementation '}
METHOD prvStart : BOOL

{attribute 'test' := 'multitest'}
{attribute 'testcasename':='Fault FB'}
{attribute 'testcategory':='Basics'}
{attribute 'testcasetimeout':='5000'}
FUNCTION_BLOCK FB_Fault_Test EXTENDS TM.Testcase_Base
VAR_INPUT
     xGetTestInfo : BOOL;
    diTestCaseIndex : DINT;
END_VAR
VAR_OUTPUT
   sTestCaseName : STRING;
    sTestCaseCategories : STRING;
    diTestCaseCount : DINT;
    diTestCaseTimeout : DINT;
    sInfo : STRING;
    eError : FB_Fault_Test_Errors;
    sError : STRING;
    eFailureMode : TM.FAILUREMODE;
END_VAR
VAR
	faultToTest : FB_Fault(name := 'Test Fault');
END_VAR

SUPER^();

{attribute 'hide'}
METHOD prvAbort : BOOL

SUPER^.prvAbort();

xAbortInProgress := FALSE;

{attribute 'hide'}
METHOD prvCyclicAction : BOOL

SUPER^.prvCyclicAction();
faultToTest.Execute();
THIS^.diTestCaseCount := 3;
CASE diTestCaseIndex OF
    0: // Test Case #0
        IF THIS^.xGetTestInfo THEN
            THIS^.sTestCaseName := 'Step 1: Check Fault is not active';
            THIS^.sTestCaseCategories := 'General';
            THIS^.diTestCaseTimeout := 3000;
			xDone := TRUE;
		ELSE
			IF NOT faultToTest.FaultActive THEN
				 xDone := TRUE;
			ELSE
				THIS^.sError := 'Fault Active before Trigger';
				xError := TRUE;
				eError := FB_Fault_Test_Errors.Fault_Active;
            	eFailureMode := TM.FAILUREMODE.AbortTestCase;
                iError := 1;
			END_IF
        END_IF
    1: // Test Case #1
        IF THIS^.xGetTestInfo THEN
            THIS^.sTestCaseName := 'Step 2: Trigger Fault';
            THIS^.sTestCaseCategories := 'General';
            THIS^.diTestCaseTimeout := 3000;
            xDone := TRUE;
		ELSE
			faultToTest.Trigger();
			IF faultToTest.FaultActive THEN
				 xDone := TRUE;
			ELSE
				THIS^.sError := 'Fault Failed to Trigger';
				xError := TRUE;
				eError := FB_Fault_Test_Errors.Fault_Not_Triggered;
				eFailureMode := TM.FAILUREMODE.AbortTestCase;
                iError := 2;
			END_IF
       END_IF

	2:	//
		IF THIS^.xGetTestInfo THEN
            THIS^.sTestCaseName := 'Step 3: Reset Fault';
            THIS^.sTestCaseCategories := 'General';
            THIS^.diTestCaseTimeout := 3000;
            xDone := TRUE;
		ELSE
			faultToTest.Ack();
			faultToTest.Execute();
			IF NOT faultToTest.FaultActive THEN
				 xDone := TRUE;
			ELSE
				THIS^.sError := 'Fault did not reset';
				xError := TRUE;
				eError := FB_Fault_Test_Errors.Fault_Not_Reset;
				eFailureMode := TM.FAILUREMODE.AbortTestCase;
                iError := 3;
			END_IF
       END_IF

    ELSE
        IF THIS^.diTestCaseIndex < 0 THEN
            THIS^.diTestCaseCount := 3;
            xDone := TRUE;
        ELSE
            THIS^.sInfo := 'Invalid test case index';
            eError := FB_Fault_Test_Errors.Fault_Not_Reset;
			xError := TRUE;
        END_IF
END_CASE

{attribute 'hide'}
METHOD prvResetOutputs : BOOL

SUPER^.prvResetOutputs();

sTestCaseName := '';
sTestCaseCategories := '';
diTestCaseCount := 0;
diTestCaseTimeout := 0;
sInfo := '';
sError := '';
eFailureMode := TM.FAILUREMODE.AbortTestCase;
eError := FB_Fault_Test_Errors.No_Error;

{attribute 'hide'}
{warning 'Add method implementation '}
METHOD prvStart : BOOL

(* ---- FB_GetTime.st ---- *)
FUNCTION_BLOCK FB_GetTime
VAR_INPUT
END_VAR
VAR_OUTPUT
    currentDateAndTime : DATE_AND_TIME;

END_VAR
VAR
    iState                    : INT;
    udiUtcTime             : UDINT;
    udiUtcTimeLocal     : UDINT;
    strTimeDate         : SYSTIMEDATE;
    strTimeDateLocal     : SYSTIMEDATE;
    dtDateTimeUTC        : DATE_AND_TIME;
    timeLeftTime        : TIME;
    timeLeftDWORD        : DWORD;
    dDateUTC            : DATE;
    todTimeOfDayUTC        : TOD;

    tSysStartTime        : TIME;
    systimeStartNano    : SYSTIME;
    udiStartTimeResult    : UDINT;

    udiResult             : UDINT;

    GetDateAndTime            : DTU.GetDateAndTime;
    SetTimeZoneInformation    : DTU.SetTimeZoneInformation;

    dtCurrent                : DATE_AND_TIME;
    dtConcated                : DATE_AND_TIME;
    //eWeekday                 : RTCLK.WEEKDAY;
    uiYear                     : UINT;
    uiMonth                     : UINT;
    uiDay                     : UINT;
    uiHour                     : UINT;
    uiMinute                 : UINT;
    uiSecond                 : UINT;

    dtuError                : DTU.ERROR;
END_VAR

CASE iState OF

    0:
        iState:= 1;

    1:  // retrieves the target date and time, including the timezone information which was set before
        GetDateAndTime( xExecute:= TRUE);
        IF GetDateAndTime.xDone THEN
            dtCurrent:= GetDateAndTime.dtDateAndTime;
            GetDateAndTime(xExecute:= FALSE);
			currentDateAndTime := dtCurrent;
            //timeLeft := TIME_TO_DT(DT_TO_TIME(targetDate) - DT_TO_TIME(dttarget));
            iState:= 2;
        END_IF
        IF GetDateAndTime.xError THEN
            GetDateAndTime(xExecute:= FALSE);
            iState:= 32767;
        END_IF

    2: (*set a spedific date and time --> returns a variable of type DATE_AND_TIME
         DateConcat --> set only date information --> returns a variable of type DATE
         TODConcat  --> set only the time information  --> returns a variable of TOD (Time of day) *)
        IF dtuError = 0 THEN
            iState := 3;
        ELSE
            iState := 32767;
        END_IF

    3:  (*a DATE_AND_TIME variable is splitted in its parts, like year, month, day etc.
            DateSplit --> the same function for a DATE variable
            TODSplit  --> the same function for a TOD variable *)

        IF dtuError = 0 THEN
            iState:= 1;
        ELSE
            iState:= 32767;
        END_IF

    32767: ; //error

END_CASE

(* ---- FB_HMIData.st ---- *)
{attribute 'FBVisuCreator'}
FUNCTION_BLOCK FB_HMIData
VAR_INPUT
	initiateCycle : BOOL;  // Initiate Cycle Pushbutton
	ackAllFaults : BOOL; // Acknowledge All Faults from HMI
	makeReady : BOOL;
	pressureBarService : ServiceCommands;
	loadPlateService : ServiceCommands;
    stopMachine : BOOL;
	{attribute 'FBVisuCreatorFormatString' := '%s'}
	version : STRING := '0.2A';
	inCycle : BOOL;
	batchEnable : BOOL;
	{attribute 'FBVisuCreatorFormatString' := '%d'}
	batchSetting : UDINT := 10;
	{attribute 'FBVisuCreatorFormatString' := '%d'}
	batchCount : UDINT;
	{attribute 'FBVisuCreatorFormatString' := '%d'}
	headCycleCount : UDINT;
	{attribute 'FBVisuCreatorFormatString' := '%1.2f'}
	pressureBarOpenDelay : REAL;
	{attribute 'FBVisuCreatorFormatString' := '%1.2f'}
	pressureBarCloseDelay : REAL;
	{attribute 'FBVisuCreatorFormatString' := '%1.2f'}
	passthroughSetting : REAL := 8.0;
	{attribute 'FBVisuCreatorFormatString' := '%1.2f'}
	passthroughActual : REAL;
	{attribute 'FBVisuCreatorFormatString' := '%1.2f'}
	lpaDwell : REAL;
	{attribute 'FBVisuCreatorFormatString' := '%1.2f'}
	hpaDwell : REAL;
	{attribute 'FBVisuCreatorFormatString' := '%1.2f'}
	sealBarDwell : REAL := 0.750;
	{attribute 'FBVisuCreatorFormatString' := '%d'}
	sealBarTemperatureSetting : UDINT;
	{attribute 'FBVisuCreatorFormatString' := '%d'}
	sealBarTemperature : UDINT;
	{attribute 'FBVisuCreatorFormatString' := '%1.2f'}
	sealFlattenerBagOpenPositionSetting : REAL;
	{attribute 'FBVisuCreatorFormatString' := '%1.2f'}
	sealFlattenerFlattenedPositionSetting : REAL;
	{attribute 'FBVisuCreatorFormatString' := '%1.2f'}
	sealFlattenerMoveInPositionSetting : REAL;
	{attribute 'FBVisuCreatorFormatString' := '%1.2f'}
	bagSkirtLength : REAL := 1.35;
	{attribute 'FBVisuCreatorFormatString' := '%1.2f'}
	bagLength : REAL := 23.5;
	{attribute 'FBVisuCreatorFormatString' := '%1.2f'}
	bagWidth : REAL := 17.5;
	{attribute 'FBVisuCreatorFormatString' := '%1.2f'}
	bagThickness : REAL := 2.5;
	{attribute 'FBVisuCreatorFormatString' := '%d'}
	bagForwardSpeed : UDINT := 55;
	{attribute 'FBVisuCreatorFormatString' := '%d'}
	bagReverseSpeed : UDINT := 3;
	{attribute 'FBVisuCreatorFormatString' := '%d'}
	printSpeed : UDINT := 6;
	{attribute 'FBVisuCreatorFormatString' := '%1.2f'}
	printLength : REAL := 8.0;
	{attribute 'FBVisuCreatorFormatString' := '%1.2f'}
	printOffset : REAL := 2.0;
	{attribute 'FBVisuCreatorFormatString' := '%d'}
	fillerCountSetting : UDINT;
	{attribute 'FBVisuCreatorFormatString' := '%d'}
	fillerCurrentCount : UDINT;
	{attribute 'FBVisuCreatorFormatString' := '%1.2f'}
	fillerDropTime : REAL;
	{attribute 'FBVisuCreatorFormatString' := '%1.2f'}
	loadPlateDelay : REAL;
	{attribute 'FBVisuCreatorFormatString' := '%1.2f'}
	loadPlateDwell : REAL := 2.5;
	exitConveyorService: ServiceCommands;
	{attribute 'FBVisuCreatorFormatString' := '%1.2f'}
	exitConveyorDwell : REAL := 9.0;
	{attribute 'FBVisuCreatorFormatString' := '%1.2f'}
	lastCycleTime : REAL;
	{attribute 'FBVisuCreatorFormatString' := '%1.2f'}
	bagDropClearanceDwell : REAL := 0.5;
	{attribute 'FBVisuCreatorFormatString' := '%1.2f'}
	averageCycleTime : REAL;
	resetAverageCycleTime : BOOL;
	{attribute 'FBVisuCreatorFormatString' := '%d'}
	bagOpenRetrySetting : UINT := 3;
	{attribute 'FBVisuCreatorFormatString' := '%d'}
	bagOpenRetryCount : UINT;
	{attribute 'FBVisuCreatorFormatString' := '%d'}
	currentJobID : INT;
	separateBeforeSeal : BOOL := TRUE;
	activateDemoMode : BOOL;
	bagOpenAssistEnable : BOOL := TRUE;
	bagOpenSensorEnable : BOOL := TRUE;
	{attribute 'FBVisuCreatorFormatString' := '%1.2f'}
	grabBagDelay : REAL := 0.5;
	{attribute 'FBVisuCreatorFormatString' := '%1.2f'}
	checkForBagOpenDelay : REAL := 1.0;
	{attribute 'FBVisuCreatorFormatString' := '%1.2f'}
	bagClearedFromFingersDelay : REAL := 0.5;
	{attribute 'FBVisuCreatorFormatString' := '%1.2f'}
	vacuumDwell : REAL := 0.5;
	(*Faults*)
	{attribute 'FBVisuCreatorFormatString' := '%s'}
	pressureBarState : STRING;
    stationValveSelection : ARRAY[1..16] OF ValveSelection := 	[ValveSelection.PressureBar,
																ValveSelection.PressureBar,
																ValveSelection.SealBar,
																ValveSelection.HPA_LPA,
																ValveSelection.LoadPlate,
																ValveSelection.BagOpenFingers,
																ValveSelection.PrintHead,
																ValveSelection.Vacuum,
																ValveSelection.SealFlattenersVerticalAxis,
																ValveSelection.LoadShelf,
																6(ValveSelection.Blank)];
    (*Counters*)
    //baggerCycles : FB_MachineCounter(name := 'Bagger Cycle Counter');
	pressureBarCycles : FB_MachineCounter(name := 'Pressure Bar Cycle Counter');
	//passthroughChanges : FB_MachineCounter(name := 'Passthrough Changes Counter');
	//loadPlateCycles : FB_MachineCounter(name := 'Load Plate Cycle Counter');
	//printerCycles : FB_MachineCounter(name := 'Printer Cycle Counter');
	//motorizedSealFlattenerCycles : FB_MachineCounter(name := 'Motorized Seal Flattener Cycles');
	//bagOpenRetryTotal : FB_MachineCounter(name := 'Bag Open Retry Totals');
	(*Info*)
	faultActive : BOOL;
	simulateAllIO : BOOL;

	(*Factoy Config*)
	bofSelection : BagOpenFingersSelection := BagOpenFingersSelection.PneumaticWithBagOpenSensors;
	bofEnable : BOOL := TRUE;
	sealFlattenersSelection : SealFlattenerSelection := SealFlattenerSelection.MotorizedSealFlatteners;
	sealFlattenersEnable : BOOL := TRUE;
	printerSelection : LabelPrinterSelection := LabelPrinterSelection.ZebraPrinter;
	printerEnable : BOOL := TRUE;
	integratedExitConveyorSelection : IntegratedConveyorSelection := IntegratedConveyorSelection.RearExit;
	integratedExitConveyorEnable : BOOL := TRUE;
	packageEjectSelection : PackageEjectionSelection := PackageEjectionSelection.RearRetractingLoadPlate;
	packageEjectEnable : BOOL := TRUE;
END_VAR
VAR_OUTPUT
END_VAR
VAR
END_VAR

(* ---- FB_InternalLogger.st ---- *)
FUNCTION_BLOCK FB_InternalLogger IMPLEMENTS IMachineLogger
VAR_INPUT
END_VAR
VAR_OUTPUT
END_VAR
VAR
	//loggedItems : ARRAY[0..500] OF FaultLogType;
	loggedItems : ARRAY[0..GLobals.MAX_LOGGED_ITEMS] OF LogMessageType;
	numOfLogEntries : UINT;
	logFull : BOOL;
	RTC : FB_GetTime();
	clearLog : BOOL;
	i : UINT;
END_VAR

//	Function Block: FB_Logger
//	Description: This is an internal logger for reference within Codesys.  It is an array that can be displayed on the TargetVisu/WebVisu
//
//	Created by: Ben Hess
//	Created Date: Tuesday, September 11, 2018

RTC();

IF clearLog THEN
	FOR i := 0 TO Globals.MAX_LOGGED_ITEMS BY 1 DO
		loggedItems[i].logMessage := '';
		loggedItems[i].logTime := DT#1970-1-1-1:0:0;
	END_FOR
	numOfLogEntries := 0;
	logFull := FALSE;
	clearLog := FALSE;
END_IF

METHOD AddLogItem
VAR_INPUT
	//category : STRING;
	message : STRING;
END_VAR

FOR i := Globals.MAX_LOGGED_ITEMS -1 TO 1 BY -1 DO
		loggedItems[i] := loggedItems[i-1];
END_FOR
//loggedItems[0].logCategory := category;
loggedItems[0].logMessage := message;
loggedItems[0].logTime := RTC.currentDateAndTime;

PROPERTY InstanceName : STRING

FUNCTION_BLOCK FB_InternalLogger IMPLEMENTS IMachineLogger
VAR_INPUT
END_VAR
VAR_OUTPUT
END_VAR
VAR
	//loggedItems : ARRAY[0..500] OF FaultLogType;
	loggedItems : ARRAY[0..GLobals.MAX_LOGGED_ITEMS] OF LogMessageType;
	numOfLogEntries : UINT;
	logFull : BOOL;
	RTC : FB_GetTime();
	clearLog : BOOL;
	i : UINT;
END_VAR

//	Function Block: FB_Logger
//	Description: This is an internal logger for reference within Codesys.  It is an array that can be displayed on the TargetVisu/WebVisu
//
//	Created by: Ben Hess
//	Created Date: Tuesday, September 11, 2018

RTC();

IF clearLog THEN
	FOR i := 0 TO Globals.MAX_LOGGED_ITEMS BY 1 DO
		loggedItems[i].logMessage := '';
		loggedItems[i].logTime := DT#1970-1-1-1:0:0;
	END_FOR
	numOfLogEntries := 0;
	logFull := FALSE;
	clearLog := FALSE;
END_IF

METHOD AddLogItem
VAR_INPUT
	//category : STRING;
	message : STRING;
END_VAR

FOR i := Globals.MAX_LOGGED_ITEMS -1 TO 1 BY -1 DO
		loggedItems[i] := loggedItems[i-1];
END_FOR
//loggedItems[0].logCategory := category;
loggedItems[0].logMessage := message;
loggedItems[0].logTime := RTC.currentDateAndTime;

PROPERTY InstanceName : STRING

(* ---- FB_IOLinkBlock.st ---- *)
{attribute 'FBVisuCreator'}
FUNCTION_BLOCK FINAL FB_IOLinkBlock EXTENDS FB_Murr16PointCFGIO
VAR_INPUT
END_VAR
VAR_OUTPUT
	iIOLinkPort4 : WORD;
	iIOLinkPort5 : WORD;
	iIOLinkPort6 : WORD;
	iIOLinkPort7 : WORD;
END_VAR
VAR
END_VAR

SUPER^();

iIOLinkPort4 :=  TO_WORD(OSCAT_BASIC.WORD_OF_BYTE(B0 := ptrEIPInputs[3], B1 := ptrEIPInputs[2]));
iIOLinkPort5 :=  TO_WORD(OSCAT_BASIC.WORD_OF_BYTE(B0 := ptrEIPInputs[5], B1 := ptrEIPInputs[4]));
iIOLinkPort6 :=  TO_WORD(OSCAT_BASIC.WORD_OF_BYTE(B0 := ptrEIPInputs[7], B1 := ptrEIPInputs[6]));
iIOLinkPort7 :=  TO_WORD(OSCAT_BASIC.WORD_OF_BYTE(B0 := ptrEIPInputs[9], B1 := ptrEIPInputs[8]));

{attribute 'FBVisuCreator'}
FUNCTION_BLOCK FINAL FB_IOLinkBlock EXTENDS FB_Murr16PointCFGIO
VAR_INPUT
END_VAR
VAR_OUTPUT
	iIOLinkPort4 : WORD;
	iIOLinkPort5 : WORD;
	iIOLinkPort6 : WORD;
	iIOLinkPort7 : WORD;
END_VAR
VAR
END_VAR

SUPER^();

iIOLinkPort4 :=  TO_WORD(OSCAT_BASIC.WORD_OF_BYTE(B0 := ptrEIPInputs[3], B1 := ptrEIPInputs[2]));
iIOLinkPort5 :=  TO_WORD(OSCAT_BASIC.WORD_OF_BYTE(B0 := ptrEIPInputs[5], B1 := ptrEIPInputs[4]));
iIOLinkPort6 :=  TO_WORD(OSCAT_BASIC.WORD_OF_BYTE(B0 := ptrEIPInputs[7], B1 := ptrEIPInputs[6]));
iIOLinkPort7 :=  TO_WORD(OSCAT_BASIC.WORD_OF_BYTE(B0 := ptrEIPInputs[9], B1 := ptrEIPInputs[8]));

(* ---- FB_LoggableBool.st ---- *)
FUNCTION_BLOCK FB_LoggableBool EXTENDS FB_BaseObject IMPLEMENTS ILoggable
VAR_INPUT
	in : BOOL;
END_VAR
VAR_OUTPUT
	Q : BOOL;
END_VAR
VAR
END_VAR

FUNCTION_BLOCK FB_LoggableBool EXTENDS FB_BaseObject IMPLEMENTS ILoggable
VAR_INPUT
	in : BOOL;
END_VAR
VAR_OUTPUT
	Q : BOOL;
END_VAR
VAR
END_VAR

(* ---- FB_MachineCounter.st ---- *)
FUNCTION_BLOCK FINAL FB_MachineCounter EXTENDS FB_BaseObject IMPLEMENTS ICounter
VAR_INPUT
END_VAR
VAR_OUTPUT
END_VAR
VAR PERSISTENT RETAIN
    count : UDINT;
END_VAR

METHOD Clear
VAR_INPUT
END_VAR

count := 0;

METHOD Increment
VAR_INPUT
END_VAR

count := count + 1;

METHOD SetCount
VAR_INPUT
	countSetting : UDINT;
END_VAR

count := countSetting;

METHOD AddToCount
VAR_INPUT
	amountToAdd : UDINT;
END_VAR

count := count + amountToAdd;

FUNCTION_BLOCK FINAL FB_MachineCounter EXTENDS FB_BaseObject IMPLEMENTS ICounter
VAR_INPUT
END_VAR
VAR_OUTPUT
END_VAR
VAR PERSISTENT RETAIN
    count : UDINT;
END_VAR

METHOD Clear
VAR_INPUT
END_VAR

count := 0;

METHOD Increment
VAR_INPUT
END_VAR

count := count + 1;

METHOD SetCount
VAR_INPUT
	countSetting : UDINT;
END_VAR

count := countSetting;

METHOD AddToCount
VAR_INPUT
	amountToAdd : UDINT;
END_VAR

count := count + amountToAdd;

(* ---- FB_MonostableMultivibrator.st ---- *)
FUNCTION_BLOCK FB_MonostableMultivibrator EXTENDS FB_BaseComponent
VAR_INPUT
END_VAR
VAR_OUTPUT
	Q : BOOL;   // Output pulse
END_VAR
VAR
	_trigger : BOOL;
	_dwellTimeInMS : UINT := 80; 	// Pulse Dwell in mS
	_delayTimeInMS : UINT; 			// Delay before Pulse in mS
	_manualOn : BOOL;
	_manualOff : BOOL;
	active : BOOL;
	dwellTimer : Standard.TON;
	delayTimer : Standard.TON;
END_VAR

SUPER^();

// HPA is on for only as long as its setpoint.

delayTimer(IN := _trigger AND NOT dwellTimer.Q, PT := UINT_TO_TIME(_delayTimeInMS));
dwellTimer(IN := delayTimer.Q AND NOT dwellTimer.Q, PT := UINT_TO_TIME(_dwellTimeInMS));

Q:= delayTimer.Q OR _manualOn;

IF dwellTimer.Q OR _reset THEN
	active := FALSE;
	_trigger := FALSE;
	_manualOn := FALSE;
	_manualOff := FALSE;
END_IF
// Reset trigger right away
// IF _trigger THEN
// 	//active := TRUE;
// 	_trigger := FALSE;
// END_IF

PROPERTY DelaySetting : UINT

METHOD Trigger
VAR_INPUT
END_VAR

_trigger := TRUE;

PROPERTY DwellSetting : UINT

METHOD ManualOff : BOOL
VAR_INPUT
END_VAR

_manualOn := FALSE;
_manualOff := TRUE;

METHOD ManualOn
VAR_INPUT
END_VAR

_manualOn := TRUE;
_manualOff := FALSE;

FUNCTION_BLOCK FB_MonostableMultivibrator EXTENDS FB_BaseComponent
VAR_INPUT
END_VAR
VAR_OUTPUT
	Q : BOOL;   // Output pulse
END_VAR
VAR
	_trigger : BOOL;
	_dwellTimeInMS : UINT := 80; 	// Pulse Dwell in mS
	_delayTimeInMS : UINT; 			// Delay before Pulse in mS
	_manualOn : BOOL;
	_manualOff : BOOL;
	active : BOOL;
	dwellTimer : Standard.TON;
	delayTimer : Standard.TON;
END_VAR

SUPER^();

// HPA is on for only as long as its setpoint.

delayTimer(IN := _trigger AND NOT dwellTimer.Q, PT := UINT_TO_TIME(_delayTimeInMS));
dwellTimer(IN := delayTimer.Q AND NOT dwellTimer.Q, PT := UINT_TO_TIME(_dwellTimeInMS));

Q:= delayTimer.Q OR _manualOn;

IF dwellTimer.Q OR _reset THEN
	active := FALSE;
	_trigger := FALSE;
	_manualOn := FALSE;
	_manualOff := FALSE;
END_IF
// Reset trigger right away
// IF _trigger THEN
// 	//active := TRUE;
// 	_trigger := FALSE;
// END_IF

PROPERTY DelaySetting : UINT

METHOD Trigger
VAR_INPUT
END_VAR

_trigger := TRUE;

PROPERTY DwellSetting : UINT

METHOD ManualOff : BOOL
VAR_INPUT
END_VAR

_manualOn := FALSE;
_manualOff := TRUE;

METHOD ManualOn
VAR_INPUT
END_VAR

_manualOn := TRUE;
_manualOff := FALSE;

(* ---- FB_MonostableMultivibrator_UnitTests.st ---- *)
{attribute 'test' := 'multitest'}
{attribute 'testcasename':='Monostable Multivibrator'}
{attribute 'testcategory':='Basics'}
{attribute 'testcasetimeout':='360000'}
FUNCTION_BLOCK FB_MonostableMultivibrator_UnitTests EXTENDS CBM.ETrigA
VAR_INPUT
     xGetTestInfo : BOOL;
    diTestCaseIndex : DINT;
END_VAR
VAR_OUTPUT
   sTestCaseName : STRING;
    sTestCaseCategories : STRING;
    diTestCaseCount : DINT;
    diTestCaseTimeout : DINT;
    sInfo : STRING;
	eError : UnitTestErrors;
    sError : STRING;
    eFailureMode : TM.FAILUREMODE;
END_VAR
VAR
	monoMulti : FB_MonostableMultivibrator(name := 'FB_MonostableMultovibrotor Under Test');
	testDwellTimer : Standard.TON;
	testPostDwellTimer : Standard.TON;
	testDelayTimer : Standard.TON;
	triggered : BOOL;
END_VAR

SUPER^();
testDwellTimer();
testPostDwellTimer();
testDelayTimer();
monoMulti();

{attribute 'hide'}
METHOD prvAbort : BOOL

SUPER^.prvAbort();

xAbortInProgress := FALSE;

{attribute 'hide'}
METHOD prvCyclicAction : BOOL

SUPER^.prvCyclicAction();
THIS^.diTestCaseCount := 5;

CASE diTestCaseIndex OF
    0: // Test Case #0
        IF THIS^.xGetTestInfo THEN
            THIS^.sTestCaseName := 'Step 1: Test Manual On';
            THIS^.sTestCaseCategories := 'General';
            THIS^.diTestCaseTimeout := 360000;
			xDone := TRUE;
		ELSE
			monoMulti.ManualOn();
			monoMulti();
			IF monoMulti.Q THEN
				 xDone := TRUE;
			ELSE
				THIS^.sError := 'Output should be on';
				xError := TRUE;
				eError := UnitTestErrors.Failure;
            	eFailureMode := TM.FAILUREMODE.AbortTestCase;
                iError := 1;
			END_IF
        END_IF
    1: // Test Case #1
        IF THIS^.xGetTestInfo THEN
            THIS^.sTestCaseName := 'Step 2: Test Manual Off';
            THIS^.sTestCaseCategories := 'General';
            THIS^.diTestCaseTimeout := 360000;
            xDone := TRUE;
		ELSE
			monoMulti.ManualOff();
			monoMulti();
			IF NOT monoMulti.Q THEN
				 xDone := TRUE;
			ELSE
				THIS^.sError := 'Output should be off';
				xError := TRUE;
				eError := UnitTestErrors.Failure;
            	eFailureMode := TM.FAILUREMODE.AbortTestCase;
                iError := 2;
			END_IF
       END_IF

	2:	//
		IF THIS^.xGetTestInfo THEN
            THIS^.sTestCaseName := 'Step 3: Start Trigger, Test Delay';
            THIS^.sTestCaseCategories := 'General';
            THIS^.diTestCaseTimeout := 360000;
            xDone := TRUE;
		ELSE
			xBusy := TRUE;
			monoMulti.DwellSetting := 2000;
			monoMulti.DelaySetting := 500;
			IF NOT triggered THEN
				monoMulti.Trigger();
				triggered := TRUE;
			END_IF

			testDelayTimer.PT := T#450MS;
			testDelayTimer.IN := TRUE;
			testDwellTimer.PT := T#1700MS;
			testDwellTimer.IN := TRUE;
			testPostDwellTimer.PT := T#2550MS;
			testPostDwellTimer.IN := TRUE;
			IF testDelayTimer.Q THEN
				IF NOT monoMulti.Q THEN
					xBusy := FALSE;
				 	xDone := TRUE;
				ELSE
					THIS^.sError := 'Output set before delay expired';
					xBusy := FALSE;
					xError := TRUE;
					eError := UnitTestErrors.Failure2;
					eFailureMode := TM.FAILUREMODE.AbortTestCase;
					iError := 3;
				END_IF
				testDelayTimer.IN := FALSE;
				triggered := FALSE;
			END_IF

       END_IF

   	3:	IF THIS^.xGetTestInfo THEN
            THIS^.sTestCaseName := 'Step 4: Test Output after delay';
            THIS^.sTestCaseCategories := 'General';
            THIS^.diTestCaseTimeout := 360000;
            xDone := TRUE;
		ELSE
			xBusy := TRUE;
			IF testDwellTimer.Q THEN
				IF monoMulti.Q THEN
				 	xDone := TRUE;
				ELSE
					THIS^.sError := 'Output not set during dwell time';
					xError := TRUE;
					eError := UnitTestErrors.Failure;
					eFailureMode := TM.FAILUREMODE.AbortTestCase;
					iError := 3;
				END_IF
				testDwellTimer.IN := FALSE;
			END_IF

       END_IF

	4:	IF THIS^.xGetTestInfo THEN
            THIS^.sTestCaseName := 'Step 5: Output off after dwell';
            THIS^.sTestCaseCategories := 'General';
            THIS^.diTestCaseTimeout := 360000;
            xDone := TRUE;
		ELSE
			xBusy := TRUE;
			IF testPostDwellTimer.Q THEN
				IF NOT monoMulti.Q THEN
				 	xDone := TRUE;
				ELSE
					THIS^.sError := Standard.CONCAT('Output still set after dwell time', TO_STRING(monoMulti.dwellTimer.ET));
					xError := TRUE;
					eError := UnitTestErrors.Failure;
					eFailureMode := TM.FAILUREMODE.AbortTestCase;
					iError := 3;
				END_IF
				testPostDwellTimer.IN := FALSE;
			END_IF
       END_IF
    ELSE
        IF THIS^.diTestCaseIndex < 0 THEN
            THIS^.diTestCaseCount := 5;
            xDone := TRUE;
        ELSE
            THIS^.sInfo := 'Invalid test case index';
            eError := UnitTestErrors.Failure;
			xError := TRUE;
        END_IF
END_CASE

{attribute 'hide'}
METHOD prvResetOutputs : BOOL

SUPER^.prvResetOutputs();

sTestCaseName := '';
sTestCaseCategories := '';
diTestCaseCount := 0;
diTestCaseTimeout := 0;
sInfo := '';
sError := '';
eFailureMode := TM.FAILUREMODE.AbortTestCase;

{attribute 'hide'}
{warning 'Add method implementation '}
METHOD prvStart : BOOL

(* ---- FB_MultiUnitTest.st ---- *)
(*
{attribute 'test' := 'multitest'}
{attribute 'testcasename':='Monostable Multivibrator'}
{attribute 'testcategory':='Basics'}
{attribute 'testcasetimeout':='360000'}
*)
FUNCTION_BLOCK FB_MultiUnitTest EXTENDS CBM.EtrigA
VAR_INPUT
	xGetTestInfo : BOOL;
    diTestCaseIndex : DINT;
END_VAR
VAR_OUTPUT
    sTestCaseName : STRING;
	sTestCaseCategories : STRING;
    diTestCaseCount : DINT;
    diTestCaseTimeout : DINT;
    sInfo : STRING;
	eError : UnitTestErrors;
    sError : STRING;
    eFailureMode : TM.FAILUREMODE;
END_VAR
VAR

END_VAR

{attribute 'hide'}
METHOD prvAbort : BOOL

SUPER^.prvAbort();

xAbortInProgress := FALSE;

{attribute 'hide'}
METHOD prvCyclicAction : BOOL

SUPER^.prvCyclicAction();

CASE diTestCaseIndex OF
    0: 	IF THIS^.xGetTestInfo THEN
            THIS^.sTestCaseName := 'Step 1: ';
            THIS^.sTestCaseCategories := 'General';
            THIS^.diTestCaseTimeout := 3000;
			xDone := TRUE;
		ELSE
			(*TEST SOMETHING HERE*)
			IF (*CONNDITION*) FALSE THEN
				 xDone := TRUE;
			ELSE
				THIS^.sError := '';
				xError := TRUE;
				eError := UnitTestErrors.Failure;
            	eFailureMode := TM.FAILUREMODE.AbortTestCase;
                iError := 1;
			END_IF
        END_IF
    1: 	IF THIS^.xGetTestInfo THEN
            THIS^.sTestCaseName := 'Step 2: ';
            THIS^.sTestCaseCategories := 'General';
            THIS^.diTestCaseTimeout := 3000;
			xDone := TRUE;
		ELSE
			(*TEST SOMETHING HERE*)
			IF (*CONNDITION*) FALSE THEN
				 xDone := TRUE;
			ELSE
				THIS^.sError := '';
				xError := TRUE;
				eError := UnitTestErrors.Failure;
            	eFailureMode := TM.FAILUREMODE.AbortTestCase;
                iError := 1;
			END_IF
        END_IF

	2: 	IF THIS^.xGetTestInfo THEN
            THIS^.sTestCaseName := 'Step 3: ';
            THIS^.sTestCaseCategories := 'General';
            THIS^.diTestCaseTimeout := 3000;
			xDone := TRUE;
		ELSE
			(*TEST SOMETHING HERE*)
			IF (*CONNDITION*) THEN
				 xDone := TRUE;
			ELSE
				THIS^.sError := '';
				xError := TRUE;
				eError := UnitTestErrors.Failure;
            	eFailureMode := TM.FAILUREMODE.AbortTestCase;
                iError := 1;
			END_IF
        END_IF

   	3: 	IF THIS^.xGetTestInfo THEN
            THIS^.sTestCaseName := 'Step 4: ';
            THIS^.sTestCaseCategories := 'General';
            THIS^.diTestCaseTimeout := 3000;
			xDone := TRUE;
		ELSE
			(*TEST SOMETHING HERE*)
			IF (*CONNDITION*) FALSE THEN
				 xDone := TRUE;
			ELSE
				THIS^.sError := '';
				xError := TRUE;
				eError := UnitTestErrors.Failure;
            	eFailureMode := TM.FAILUREMODE.AbortTestCase;
                iError := 1;
			END_IF
        END_IF

	4: 	IF THIS^.xGetTestInfo THEN
            THIS^.sTestCaseName := 'Step 5: ';
            THIS^.sTestCaseCategories := 'General';
            THIS^.diTestCaseTimeout := 3000;
			xDone := TRUE;
		ELSE
			(*TEST SOMETHING HERE*)
			IF (*CONNDITION*) FALSE THEN
				 xDone := TRUE;
			ELSE
				THIS^.sError := '';
				xError := TRUE;
				eError := UnitTestErrors.Failure;
            	eFailureMode := TM.FAILUREMODE.AbortTestCase;
                iError := 1;
			END_IF
        END_IF

	5: 	IF THIS^.xGetTestInfo THEN
            THIS^.sTestCaseName := 'Step 6: ';
            THIS^.sTestCaseCategories := 'General';
            THIS^.diTestCaseTimeout := 3000;
			xDone := TRUE;
		ELSE
			(*TEST SOMETHING HERE*)
			IF (*CONNDITION*) FALSE THEN
				 xDone := TRUE;
			ELSE
				THIS^.sError := '';
				xError := TRUE;
				eError := UnitTestErrors.Failure;
            	eFailureMode := TM.FAILUREMODE.AbortTestCase;
                iError := 1;
			END_IF
        END_IF

	6: 	IF THIS^.xGetTestInfo THEN
            THIS^.sTestCaseName := 'Step 7: ';
            THIS^.sTestCaseCategories := 'General';
            THIS^.diTestCaseTimeout := 3000;
			xDone := TRUE;
		ELSE
			(*TEST SOMETHING HERE*)
			IF (*CONNDITION*) FALSE THEN
				 xDone := TRUE;
			ELSE
				THIS^.sError := '';
				xError := TRUE;
				eError := UnitTestErrors.Failure;
            	eFailureMode := TM.FAILUREMODE.AbortTestCase;
                iError := 1;
			END_IF
        END_IF
    ELSE
        IF THIS^.diTestCaseIndex < 0 THEN
            THIS^.diTestCaseCount := 7;
            xDone := TRUE;
        ELSE
            THIS^.sInfo := 'Invalid test case index';
            eError := UnitTestErrors.Failure;
			xError := TRUE;
        END_IF
END_CASE

{attribute 'hide'}
METHOD prvResetOutputs : BOOL

SUPER^.prvResetOutputs();

sTestCaseName := '';
sTestCaseCategories := '';
diTestCaseCount := 0;
diTestCaseTimeout := 0;
sInfo := '';
sError := '';
eFailureMode := TM.FAILUREMODE.AbortTestCase;

{attribute 'hide'}
METHOD prvStart : BOOL

(*
{attribute 'test' := 'multitest'}
{attribute 'testcasename':='Monostable Multivibrator'}
{attribute 'testcategory':='Basics'}
{attribute 'testcasetimeout':='360000'}
*)
FUNCTION_BLOCK FB_MultiUnitTest EXTENDS CBM.EtrigA
VAR_INPUT
	xGetTestInfo : BOOL;
    diTestCaseIndex : DINT;
END_VAR
VAR_OUTPUT
    sTestCaseName : STRING;
	sTestCaseCategories : STRING;
    diTestCaseCount : DINT;
    diTestCaseTimeout : DINT;
    sInfo : STRING;
	eError : UnitTestErrors;
    sError : STRING;
    eFailureMode : TM.FAILUREMODE;
END_VAR
VAR

END_VAR

{attribute 'hide'}
METHOD prvAbort : BOOL

SUPER^.prvAbort();

xAbortInProgress := FALSE;

{attribute 'hide'}
METHOD prvCyclicAction : BOOL

SUPER^.prvCyclicAction();

CASE diTestCaseIndex OF
    0: 	IF THIS^.xGetTestInfo THEN
            THIS^.sTestCaseName := 'Step 1: ';
            THIS^.sTestCaseCategories := 'General';
            THIS^.diTestCaseTimeout := 3000;
			xDone := TRUE;
		ELSE
			(*TEST SOMETHING HERE*)
			IF (*CONNDITION*) FALSE THEN
				 xDone := TRUE;
			ELSE
				THIS^.sError := '';
				xError := TRUE;
				eError := UnitTestErrors.Failure;
            	eFailureMode := TM.FAILUREMODE.AbortTestCase;
                iError := 1;
			END_IF
        END_IF
    1: 	IF THIS^.xGetTestInfo THEN
            THIS^.sTestCaseName := 'Step 2: ';
            THIS^.sTestCaseCategories := 'General';
            THIS^.diTestCaseTimeout := 3000;
			xDone := TRUE;
		ELSE
			(*TEST SOMETHING HERE*)
			IF (*CONNDITION*) FALSE THEN
				 xDone := TRUE;
			ELSE
				THIS^.sError := '';
				xError := TRUE;
				eError := UnitTestErrors.Failure;
            	eFailureMode := TM.FAILUREMODE.AbortTestCase;
                iError := 1;
			END_IF
        END_IF

	2: 	IF THIS^.xGetTestInfo THEN
            THIS^.sTestCaseName := 'Step 3: ';
            THIS^.sTestCaseCategories := 'General';
            THIS^.diTestCaseTimeout := 3000;
			xDone := TRUE;
		ELSE
			(*TEST SOMETHING HERE*)
			IF (*CONNDITION*) THEN
				 xDone := TRUE;
			ELSE
				THIS^.sError := '';
				xError := TRUE;
				eError := UnitTestErrors.Failure;
            	eFailureMode := TM.FAILUREMODE.AbortTestCase;
                iError := 1;
			END_IF
        END_IF

   	3: 	IF THIS^.xGetTestInfo THEN
            THIS^.sTestCaseName := 'Step 4: ';
            THIS^.sTestCaseCategories := 'General';
            THIS^.diTestCaseTimeout := 3000;
			xDone := TRUE;
		ELSE
			(*TEST SOMETHING HERE*)
			IF (*CONNDITION*) FALSE THEN
				 xDone := TRUE;
			ELSE
				THIS^.sError := '';
				xError := TRUE;
				eError := UnitTestErrors.Failure;
            	eFailureMode := TM.FAILUREMODE.AbortTestCase;
                iError := 1;
			END_IF
        END_IF

	4: 	IF THIS^.xGetTestInfo THEN
            THIS^.sTestCaseName := 'Step 5: ';
            THIS^.sTestCaseCategories := 'General';
            THIS^.diTestCaseTimeout := 3000;
			xDone := TRUE;
		ELSE
			(*TEST SOMETHING HERE*)
			IF (*CONNDITION*) FALSE THEN
				 xDone := TRUE;
			ELSE
				THIS^.sError := '';
				xError := TRUE;
				eError := UnitTestErrors.Failure;
            	eFailureMode := TM.FAILUREMODE.AbortTestCase;
                iError := 1;
			END_IF
        END_IF

	5: 	IF THIS^.xGetTestInfo THEN
            THIS^.sTestCaseName := 'Step 6: ';
            THIS^.sTestCaseCategories := 'General';
            THIS^.diTestCaseTimeout := 3000;
			xDone := TRUE;
		ELSE
			(*TEST SOMETHING HERE*)
			IF (*CONNDITION*) FALSE THEN
				 xDone := TRUE;
			ELSE
				THIS^.sError := '';
				xError := TRUE;
				eError := UnitTestErrors.Failure;
            	eFailureMode := TM.FAILUREMODE.AbortTestCase;
                iError := 1;
			END_IF
        END_IF

	6: 	IF THIS^.xGetTestInfo THEN
            THIS^.sTestCaseName := 'Step 7: ';
            THIS^.sTestCaseCategories := 'General';
            THIS^.diTestCaseTimeout := 3000;
			xDone := TRUE;
		ELSE
			(*TEST SOMETHING HERE*)
			IF (*CONNDITION*) FALSE THEN
				 xDone := TRUE;
			ELSE
				THIS^.sError := '';
				xError := TRUE;
				eError := UnitTestErrors.Failure;
            	eFailureMode := TM.FAILUREMODE.AbortTestCase;
                iError := 1;
			END_IF
        END_IF
    ELSE
        IF THIS^.diTestCaseIndex < 0 THEN
            THIS^.diTestCaseCount := 7;
            xDone := TRUE;
        ELSE
            THIS^.sInfo := 'Invalid test case index';
            eError := UnitTestErrors.Failure;
			xError := TRUE;
        END_IF
END_CASE

{attribute 'hide'}
METHOD prvResetOutputs : BOOL

SUPER^.prvResetOutputs();

sTestCaseName := '';
sTestCaseCategories := '';
diTestCaseCount := 0;
diTestCaseTimeout := 0;
sInfo := '';
sError := '';
eFailureMode := TM.FAILUREMODE.AbortTestCase;

{attribute 'hide'}
METHOD prvStart : BOOL

(* ---- FB_Murr16PointCFGIO.st ---- *)
{attribute 'FBVisuCreator'}
FUNCTION_BLOCK FB_Murr16PointCFGIO EXTENDS FB_BaseObject
VAR_INPUT
	ptrEIPInputs : POINTER TO BYTE;	// Pointer to starting word of EIP Inputs for the I/O Image
    ptrEIPOutputs : POINTER TO BYTE;	// Pointer to starting word of EIP Outputs for the I/O Image

	oPort0Pin2 : BOOL;
	oPort0Pin4 : BOOL;
	oPort1Pin2 : BOOL;
	oPort1Pin4 : BOOL;
	oPort2Pin2 : BOOL;
	oPort2Pin4 : BOOL;
	oPort3Pin2 : BOOL;
	oPort3Pin4 : BOOL;
	oPort4Pin2 : BOOL;
	oPort4Pin4 : BOOL;
	oPort5Pin2 : BOOL;
	oPort5Pin4 : BOOL;
	oPort6Pin2 : BOOL;
	oPort6Pin4 : BOOL;
	oPort7Pin2 : BOOL;
	oPort7Pin4 : BOOL;
END_VAR
VAR_OUTPUT
	iPort0Pin2 : BOOL;
	iPort0Pin4 : BOOL;
	iPort1Pin2 : BOOL;
	iPort1Pin4 : BOOL;
	iPort2Pin2 : BOOL;
	iPort2Pin4 : BOOL;
	iPort3Pin2 : BOOL;
	iPort3Pin4 : BOOL;
	iPort4Pin2 : BOOL;
	iPort4Pin4 : BOOL;
	iPort5Pin2 : BOOL;
	iPort5Pin4 : BOOL;
	iPort6Pin2 : BOOL;
	iPort6Pin4 : BOOL;
	iPort7Pin2 : BOOL;
	iPort7Pin4 : BOOL;
END_VAR
VAR_IN_OUT
END_VAR
VAR
END_VAR

iPort0Pin2 := ptrEIPInputs[1].0;
iPort0Pin4 := ptrEIPInputs[0].0;
iPort1Pin2 := ptrEIPInputs[1].1;
iPort1Pin4 := ptrEIPInputs[0].1;
iPort2Pin2 := ptrEIPInputs[1].2;
iPort2Pin4 := ptrEIPInputs[0].2;
iPort3Pin2 := ptrEIPInputs[1].3;
iPort3Pin4 := ptrEIPInputs[0].3;
iPort4Pin2 := ptrEIPInputs[1].4;
iPort4Pin4 := ptrEIPInputs[0].4;
iPort5Pin2 := ptrEIPInputs[1].5;
iPort5Pin4 := ptrEIPInputs[0].5;
iPort6Pin2 := ptrEIPInputs[1].6;
iPort6Pin4 := ptrEIPInputs[0].6;
iPort7Pin2 := ptrEIPInputs[1].7;
iPort7Pin4 := ptrEIPInputs[0].7;

ptrEIPOutputs[1].0 := oPort0Pin2;
ptrEIPOutputs[0].0 := oPort0Pin4;
ptrEIPOutputs[1].1 := oPort1Pin2;
ptrEIPOutputs[0].1 := oPort1Pin4;
ptrEIPOutputs[1].2 := oPort2Pin2;
ptrEIPOutputs[0].2 := oPort2Pin4;
ptrEIPOutputs[1].3 := oPort3Pin2;
ptrEIPOutputs[0].3 := oPort3Pin4;
ptrEIPOutputs[1].4 := oPort4Pin2;
ptrEIPOutputs[0].4 := oPort4Pin4;
ptrEIPOutputs[1].5 := oPort5Pin2;
ptrEIPOutputs[0].5 := oPort5Pin4;
ptrEIPOutputs[1].6 := oPort6Pin2;
ptrEIPOutputs[0].6 := oPort6Pin4;
ptrEIPOutputs[1].7 := oPort7Pin2;
ptrEIPOutputs[0].7 := oPort7Pin4;

{attribute 'FBVisuCreator'}
FUNCTION_BLOCK FB_Murr16PointCFGIO EXTENDS FB_BaseObject
VAR_INPUT
	ptrEIPInputs : POINTER TO BYTE;	// Pointer to starting word of EIP Inputs for the I/O Image
    ptrEIPOutputs : POINTER TO BYTE;	// Pointer to starting word of EIP Outputs for the I/O Image

	oPort0Pin2 : BOOL;
	oPort0Pin4 : BOOL;
	oPort1Pin2 : BOOL;
	oPort1Pin4 : BOOL;
	oPort2Pin2 : BOOL;
	oPort2Pin4 : BOOL;
	oPort3Pin2 : BOOL;
	oPort3Pin4 : BOOL;
	oPort4Pin2 : BOOL;
	oPort4Pin4 : BOOL;
	oPort5Pin2 : BOOL;
	oPort5Pin4 : BOOL;
	oPort6Pin2 : BOOL;
	oPort6Pin4 : BOOL;
	oPort7Pin2 : BOOL;
	oPort7Pin4 : BOOL;
END_VAR
VAR_OUTPUT
	iPort0Pin2 : BOOL;
	iPort0Pin4 : BOOL;
	iPort1Pin2 : BOOL;
	iPort1Pin4 : BOOL;
	iPort2Pin2 : BOOL;
	iPort2Pin4 : BOOL;
	iPort3Pin2 : BOOL;
	iPort3Pin4 : BOOL;
	iPort4Pin2 : BOOL;
	iPort4Pin4 : BOOL;
	iPort5Pin2 : BOOL;
	iPort5Pin4 : BOOL;
	iPort6Pin2 : BOOL;
	iPort6Pin4 : BOOL;
	iPort7Pin2 : BOOL;
	iPort7Pin4 : BOOL;
END_VAR
VAR_IN_OUT
END_VAR
VAR
END_VAR

iPort0Pin2 := ptrEIPInputs[1].0;
iPort0Pin4 := ptrEIPInputs[0].0;
iPort1Pin2 := ptrEIPInputs[1].1;
iPort1Pin4 := ptrEIPInputs[0].1;
iPort2Pin2 := ptrEIPInputs[1].2;
iPort2Pin4 := ptrEIPInputs[0].2;
iPort3Pin2 := ptrEIPInputs[1].3;
iPort3Pin4 := ptrEIPInputs[0].3;
iPort4Pin2 := ptrEIPInputs[1].4;
iPort4Pin4 := ptrEIPInputs[0].4;
iPort5Pin2 := ptrEIPInputs[1].5;
iPort5Pin4 := ptrEIPInputs[0].5;
iPort6Pin2 := ptrEIPInputs[1].6;
iPort6Pin4 := ptrEIPInputs[0].6;
iPort7Pin2 := ptrEIPInputs[1].7;
iPort7Pin4 := ptrEIPInputs[0].7;

ptrEIPOutputs[1].0 := oPort0Pin2;
ptrEIPOutputs[0].0 := oPort0Pin4;
ptrEIPOutputs[1].1 := oPort1Pin2;
ptrEIPOutputs[0].1 := oPort1Pin4;
ptrEIPOutputs[1].2 := oPort2Pin2;
ptrEIPOutputs[0].2 := oPort2Pin4;
ptrEIPOutputs[1].3 := oPort3Pin2;
ptrEIPOutputs[0].3 := oPort3Pin4;
ptrEIPOutputs[1].4 := oPort4Pin2;
ptrEIPOutputs[0].4 := oPort4Pin4;
ptrEIPOutputs[1].5 := oPort5Pin2;
ptrEIPOutputs[0].5 := oPort5Pin4;
ptrEIPOutputs[1].6 := oPort6Pin2;
ptrEIPOutputs[0].6 := oPort6Pin4;
ptrEIPOutputs[1].7 := oPort7Pin2;
ptrEIPOutputs[0].7 := oPort7Pin4;

(* ---- FB_Murr56691_IP20.st ---- *)
{attribute 'FBVisuCreator'}
FUNCTION_BLOCK FB_Murr56691_IP20 EXTENDS FB_BaseObject
VAR_INPUT
	ptrEIPInputs : POINTER TO BYTE;	// Pointer to starting word of EIP Inputs for the I/O Image
    ptrEIPOutputs : POINTER TO BYTE;	// Pointer to starting word of EIP Outputs for the I/O Image

	oX100 : BOOL;
	oX101 : BOOL;
	oX102 : BOOL;
	oX103 : BOOL;
	oX104 : BOOL;
	oX105 : BOOL;
	oX106 : BOOL;
	oX107 : BOOL;
END_VAR
VAR_OUTPUT

	iX000 : BOOL;
	iX001 : BOOL;
	iX002 : BOOL;
	iX003 : BOOL;
	iX004 : BOOL;
	iX005 : BOOL;
	iX006 : BOOL;
	iX007 : BOOL;

	iX100 : BOOL;
	iX101 : BOOL;
	iX102 : BOOL;
	iX103 : BOOL;
	iX104 : BOOL;
	iX105 : BOOL;
	iX106 : BOOL;
	iX107 : BOOL;
END_VAR
VAR_IN_OUT
END_VAR
VAR
END_VAR
//	Function Block: FB_Murr56691_IP20
//	Description: Abstracts a Murr 56691 IP20 I/O Block
//
//	Created by: Ben Hess
//	Created Date: Friday, October 19, 2018

iX100 := ptrEIPInputs[0].0;
iX101 := ptrEIPInputs[0].1;
iX102 := ptrEIPInputs[0].2;
iX103 := ptrEIPInputs[0].3;
iX104 := ptrEIPInputs[0].4;
iX105 := ptrEIPInputs[0].5;
iX106 := ptrEIPInputs[0].6;
iX107 := ptrEIPInputs[0].7;

iX000 := ptrEIPInputs[1].0;
iX001 := ptrEIPInputs[1].1;
iX002 := ptrEIPInputs[1].2;
iX003 := ptrEIPInputs[1].3;
iX004 := ptrEIPInputs[1].4;
iX005 := ptrEIPInputs[1].5;
iX006 := ptrEIPInputs[1].6;
iX007 := ptrEIPInputs[1].7;

ptrEIPOutputs[0].0 := oX100;
ptrEIPOutputs[0].1 := oX101;
ptrEIPOutputs[0].2 := oX102;
ptrEIPOutputs[0].3 := oX103;
ptrEIPOutputs[0].4 := oX104;
ptrEIPOutputs[0].5 := oX105;
ptrEIPOutputs[0].6 := oX106;
ptrEIPOutputs[0].7 := oX107;

{attribute 'FBVisuCreator'}
FUNCTION_BLOCK FB_Murr56691_IP20 EXTENDS FB_BaseObject
VAR_INPUT
	ptrEIPInputs : POINTER TO BYTE;	// Pointer to starting word of EIP Inputs for the I/O Image
    ptrEIPOutputs : POINTER TO BYTE;	// Pointer to starting word of EIP Outputs for the I/O Image

	oX100 : BOOL;
	oX101 : BOOL;
	oX102 : BOOL;
	oX103 : BOOL;
	oX104 : BOOL;
	oX105 : BOOL;
	oX106 : BOOL;
	oX107 : BOOL;
END_VAR
VAR_OUTPUT

	iX000 : BOOL;
	iX001 : BOOL;
	iX002 : BOOL;
	iX003 : BOOL;
	iX004 : BOOL;
	iX005 : BOOL;
	iX006 : BOOL;
	iX007 : BOOL;

	iX100 : BOOL;
	iX101 : BOOL;
	iX102 : BOOL;
	iX103 : BOOL;
	iX104 : BOOL;
	iX105 : BOOL;
	iX106 : BOOL;
	iX107 : BOOL;
END_VAR
VAR_IN_OUT
END_VAR
VAR
END_VAR
//	Function Block: FB_Murr56691_IP20
//	Description: Abstracts a Murr 56691 IP20 I/O Block
//
//	Created by: Ben Hess
//	Created Date: Friday, October 19, 2018

iX100 := ptrEIPInputs[0].0;
iX101 := ptrEIPInputs[0].1;
iX102 := ptrEIPInputs[0].2;
iX103 := ptrEIPInputs[0].3;
iX104 := ptrEIPInputs[0].4;
iX105 := ptrEIPInputs[0].5;
iX106 := ptrEIPInputs[0].6;
iX107 := ptrEIPInputs[0].7;

iX000 := ptrEIPInputs[1].0;
iX001 := ptrEIPInputs[1].1;
iX002 := ptrEIPInputs[1].2;
iX003 := ptrEIPInputs[1].3;
iX004 := ptrEIPInputs[1].4;
iX005 := ptrEIPInputs[1].5;
iX006 := ptrEIPInputs[1].6;
iX007 := ptrEIPInputs[1].7;

ptrEIPOutputs[0].0 := oX100;
ptrEIPOutputs[0].1 := oX101;
ptrEIPOutputs[0].2 := oX102;
ptrEIPOutputs[0].3 := oX103;
ptrEIPOutputs[0].4 := oX104;
ptrEIPOutputs[0].5 := oX105;
ptrEIPOutputs[0].6 := oX106;
ptrEIPOutputs[0].7 := oX107;

(* ---- FB_MurrMaster.st ---- *)
FUNCTION_BLOCK FB_MurrMaster EXTENDS FB_BaseObject
VAR_INPUT
	ptrEIPInputs : POINTER TO BYTE;	// Pointer to starting word of EIP Inputs for the I/O Image
    ptrEIPOutputs : POINTER TO BYTE;	// Pointer to starting word of EIP Outputs for the I/O Image
END_VAR
VAR_OUTPUT
	headIONode : FB_IOLinkBlock(name := 'Head Block');
	frontGuardIONode : FB_Murr16PointCFGIO(name := 'Front Guard Block');
	dischargeIONode : FB_Murr16PointCFGIO(name := 'Discharge Block');
	printerIONode : FB_Murr56691_IP20(name := 'Printer Block');
END_VAR
VAR
END_VAR
VAR (*Faults*)
	commFail : FB_Fault(name := CONCAT(_prefix,  'Communication Failure'));
END_VAR
// Head IO Node, offset of 0 for I/O
headIONode(ptrEIPInputs := ptrEIPInputs, ptrEIPOutputs := ptrEIPOutputs);
frontGuardIONode(ptrEIPInputs := ADR(ptrEIPInputs[30]), ptrEIPOutputs := ADR(ptrEIPOutputs[30]));
dischargeIONode(ptrEIPInputs := ADR(ptrEIPInputs[32]), ptrEIPOutputs := ADR(ptrEIPOutputs[32]));
printerIONode(ptrEIPInputs := ADR(ptrEIPInputs[34]), ptrEIPOutputs := ADR(ptrEIPOutputs[34]));
{region 'Alarms'}

{endregion}

(* ---- FB_PackMLStates.st ---- *)
FUNCTION_BLOCK FB_PackMLStates EXTENDS FB_BaseObject IMPLEMENTS IPackMLStates, IAllObjects
VAR_INPUT
END_VAR
VAR_OUTPUT
END_VAR
VAR
	_abortingDone : BOOL;
	_clearingDone : BOOL;
	_completingDone : BOOL;
	_holdingDone : BOOL;
	_resettingDone : BOOL;
	_startingDone : BOOL;
	_unholdingDone : BOOL;
	_stoppingDone : BOOL;
END_VAR

PROPERTY AbortingDone : BOOL

PROPERTY ClearingDone : BOOL

PROPERTY CompletingDone : BOOL

PROPERTY HoldingDone : BOOL

PROPERTY ResettingDone : BOOL

PROPERTY StartingDone : BOOL

PROPERTY UnholdingDone : BOOL

METHOD Aborting

_abortingDone := TRUE;

METHOD Clearing

_clearingDone := TRUE;

METHOD Stopped

_clearingDone := FALSE;

METHOD Idle

_resettingDone := FALSE;

METHOD Starting

_startingDone := TRUE;

METHOD Executing

METHOD Aborted

_abortingDone := FALSE;

METHOD Stopping

_stoppingDone := TRUE;

METHOD Resetting

_resettingDone := TRUE;

METHOD Held

_holdingDone := FALSE;

METHOD Holding

_holdingDone := TRUE;

METHOD UnHolding

_unholdingDone := TRUE;

METHOD Complete

_completingDone := FALSE;

METHOD Completing

_completingDone := TRUE;

PROPERTY StoppingDone : BOOL

(* ---- FB_PhysicalAnalogInput.st ---- *)
FUNCTION_BLOCK FB_PhysicalAnalogInput EXTENDS FB_BaseObject IMPLEMENTS IExecuteAutomatically, ILoggable
VAR_INPUT
	in : REFERENCE TO WORD;		// Raw Analog Input
	enableLogging : BOOL;		// Enable logging
	logDeadband : INT;			// Deadband to log changes
END_VAR
VAR_OUTPUT
	RawValue : WORD;
END_VAR
VAR
	logged : BOOL;
	loggedValue : INT;
END_VAR

METHOD Execute
VAR_INPUT
END_VAR

VAR

END_VAR
IF __ISVALIDREF(in) THEN
	RawValue := in;
END_IF

IF TO_INT(RawValue) < (loggedValue - logDeadband) OR TO_INT(RawValue) > (loggedValue + logDeadband) THEN
	logged := FALSE;
END_IF

IF NOT logged AND enableLogging THEN
    _logger.AddLogItem(CONCAT(_prefix, TO_STRING(RawValue)));
	loggedValue := TO_INT(RawValue);
	logged := TRUE;
END_IF

FUNCTION_BLOCK FB_PhysicalAnalogInput EXTENDS FB_BaseObject IMPLEMENTS IExecuteAutomatically, ILoggable
VAR_INPUT
	in : REFERENCE TO WORD;		// Raw Analog Input
	enableLogging : BOOL;		// Enable logging
	logDeadband : INT;			// Deadband to log changes
END_VAR
VAR_OUTPUT
	RawValue : WORD;
END_VAR
VAR
	logged : BOOL;
	loggedValue : INT;
END_VAR

METHOD Execute
VAR_INPUT
END_VAR

VAR

END_VAR
IF __ISVALIDREF(in) THEN
	RawValue := in;
END_IF

IF TO_INT(RawValue) < (loggedValue - logDeadband) OR TO_INT(RawValue) > (loggedValue + logDeadband) THEN
	logged := FALSE;
END_IF

IF NOT logged AND enableLogging THEN
    _logger.AddLogItem(CONCAT(_prefix, TO_STRING(RawValue)));
	loggedValue := TO_INT(RawValue);
	logged := TRUE;
END_IF

(* ---- FB_PhysicalDigitalInput.st ---- *)
{attribute 'io_function_block'}
FUNCTION_BLOCK FB_PhysicalDigitalInput EXTENDS FB_BaseObject IMPLEMENTS IExecuteAutomatically
VAR_INPUT
	in : REFERENCE TO BOOL;
	simulate : BOOL;
	simValue : BOOL;
	debounceEnable : BOOL;	//
	debounceTime : REAL := 50.0;		// Debounce time in MS
END_VAR
VAR_OUTPUT
	Active : BOOL;
	OSR : BOOL;
	OSF : BOOL;
END_VAR
VAR
	debounceTimer : TON;
	inputONS : FB_ONS();
END_VAR

METHOD Execute
VAR_INPUT
END_VAR

IF NOT __ISVALIDREF(in) THEN
	RETURN;
END_IF

debounceTimer(IN := (in AND NOT simulate) OR (simulate AND simValue) AND debounceEnable, PT := REAL_TO_TIME(debounceTime * 1000));
inputONS();

IF debounceEnable THEN
	Active := debounceTimer.Q;
ELSE
	IF simulate THEN
		Active := simValue;
		inputONS.CLK := simValue;
	ELSE
		Active := in;
		inputONS.CLK := in;

	END_IF
END_IF

IF inputONS.OSR THEN
    _logger.AddLogItem(CONCAT(_prefix, 'On'));
END_IF

IF inputONS.OSF THEN
    _logger.AddLogItem(CONCAT(_prefix, 'Off'));
END_IF

{attribute 'monitoring' := 'variable'}
PROPERTY IsOn : BOOL

{attribute 'monitoring' := 'variable'}
PROPERTY IsOff : BOOL

{attribute 'io_function_block'}
FUNCTION_BLOCK FB_PhysicalDigitalInput EXTENDS FB_BaseObject IMPLEMENTS IExecuteAutomatically
VAR_INPUT
	in : REFERENCE TO BOOL;
	simulate : BOOL;
	simValue : BOOL;
	debounceEnable : BOOL;	//
	debounceTime : REAL := 50.0;		// Debounce time in MS
END_VAR
VAR_OUTPUT
	Active : BOOL;
	OSR : BOOL;
	OSF : BOOL;
END_VAR
VAR
	debounceTimer : TON;
	inputONS : FB_ONS();
END_VAR

METHOD Execute
VAR_INPUT
END_VAR

IF NOT __ISVALIDREF(in) THEN
	RETURN;
END_IF

debounceTimer(IN := (in AND NOT simulate) OR (simulate AND simValue) AND debounceEnable, PT := REAL_TO_TIME(debounceTime * 1000));
inputONS();

IF debounceEnable THEN
	Active := debounceTimer.Q;
ELSE
	IF simulate THEN
		Active := simValue;
		inputONS.CLK := simValue;
	ELSE
		Active := in;
		inputONS.CLK := in;

	END_IF
END_IF

IF inputONS.OSR THEN
    _logger.AddLogItem(CONCAT(_prefix, 'On'));
END_IF

IF inputONS.OSF THEN
    _logger.AddLogItem(CONCAT(_prefix, 'Off'));
END_IF

{attribute 'monitoring' := 'variable'}
PROPERTY IsOn : BOOL

{attribute 'monitoring' := 'variable'}
PROPERTY IsOff : BOOL

(* ---- FB_PhysicalDigitalOutput.st ---- *)
FUNCTION_BLOCK FB_PhysicalDigitalOutput EXTENDS FB_BaseObject IMPLEMENTS ILoggable, ISimulateable
VAR_INPUT
	refOutput : REFERENCE TO BOOL; //  Reference to physical output

END_VAR
VAR_OUTPUT
	Q : BOOL;		// Logical inidcation of output
END_VAR
VAR
	outputONS : FB_ONS;
	_simulate : BOOL;	// Simulate output - do not trigger actual physical output
END_VAR
VAR_IN_OUT

END_VAR

METHOD Execute
VAR_INPUT
END_VAR

outputONS(CLK := Q);

IF __ISVALIDREF(refoutput) THEN
	IF _simulate THEN
		refOutput := FALSE;
	ELSE
		refOutput := Q;
	END_IF
END_IF

IF outputONS.OSR THEN
    _logger.AddLogItem(CONCAT(_prefix, 'On'));
END_IF

IF outputONS.OSF THEN
    _logger.AddLogItem(CONCAT(_prefix, 'Off'));
END_IF

METHOD TurnOff
VAR_INPUT
END_VAR

Q := FALSE;
Execute();

METHOD TurnOn
VAR_INPUT
END_VAR

Q := TRUE;
Execute();

PROPERTY Simulate : BOOL
